LIN {X 0,Y 526.287,Z 607.372,A -85,B 0,C 180,E1 -4788.6,E2 -4788.6} C_VEL
LIN {X 0,Y 526.834,Z 594.37,A -85,B 0,C 180,E1 -4789.583,E2 -4789.583} C_VEL
LIN {X 0,Y 527.395,Z 580.497,A -85,B 0,C 180,E1 -4790.475,E2 -4790.475} C_VEL
LIN {X 0,Y 528.125,Z 564.209,A -85,B 0,C 180,E1 -4791.327,E2 -4791.327} C_VEL
LIN {X 0,Y 528.573,Z 550.297,A -85,B 0,C 180,E1 -4791.908,E2 -4791.908} C_VEL
LIN {X 0,Y 529.049,Z 533.497,A -85,B 0,C 180,E1 -4792.453,E2 -4792.453} C_VEL
LIN {X 0,Y 529.379,Z 517.227,A -85,B 0,C 180,E1 -4792.824,E2 -4792.824} C_VEL
LIN {X 0,Y 530.896,Z 327.244,A -85,B 0,C 180,E1 -4795.531,E2 -4795.531} C_VEL
LIN {X 0,Y 530.306,Z 322.417,A -85,B 0,C 180,E1 -4795.632,E2 -4795.632} C_VEL
LIN {X 0,Y 528.19,Z 310.861,A -85,B 0,C 180,E1 -4795.923,E2 -4795.923} C_VEL
LIN {X 0,Y 529.061,Z 286.972,A -85,B 0,C 180,E1 -4798.171,E2 -4798.171} C_VEL
LIN {X 0,Y 524.52,Z 271.582,A -85,B 0,C 180,E1 -4799.941,E2 -4799.941} C_VEL
LIN {X 0,Y 523.928,Z 269.536,A -85,B 0,C 180,E1 -4800.2,E2 -4800.2} C_VEL
LIN {X 0,Y 523.939,Z 269.532,A -85,B 0,C 180,E1 -4803.364,E2 -4803.364} C_VEL
LIN {X 0,Y 523.901,Z 269.535,A -85,B 0,C 180,E1 -4806.401,E2 -4806.401} C_VEL
LIN {X 0,Y 523.92,Z 269.539,A -85,B 0,C 180,E1 -4809.084,E2 -4809.084} C_VEL
LIN {X 0,Y 523.955,Z 269.527,A -85,B 0,C 180,E1 -4812.118,E2 -4812.118} C_VEL
LIN {X 0,Y 523.952,Z 269.534,A -85,B 0,C 180,E1 -4815.309,E2 -4815.309} C_VEL
LIN {X 0,Y 523.959,Z 269.526,A -85,B 0,C 180,E1 -4818.689,E2 -4818.689} C_VEL
LIN {X 0,Y 523.913,Z 269.531,A -85,B 0,C 180,E1 -4821.898,E2 -4821.898} C_VEL
LIN {X 0,Y 523.933,Z 269.533,A -85,B 0,C 180,E1 -4824.909,E2 -4824.909} C_VEL
LIN {X 0,Y 523.932,Z 269.532,A -85,B 0,C 180,E1 -4827.68,E2 -4827.68} C_VEL
LIN {X 0,Y 523.951,Z 269.528,A -85,B 0,C 180,E1 -4830.676,E2 -4830.676} C_VEL
LIN {X 0,Y 523.971,Z 269.527,A -85,B 0,C 180,E1 -4833.729,E2 -4833.729} C_VEL
LIN {X 0,Y 523.934,Z 269.529,A -85,B 0,C 180,E1 -4836.271,E2 -4836.271} C_VEL
LIN {X 0,Y 523.943,Z 269.531,A -85,B 0,C 180,E1 -4838.767,E2 -4838.767} C_VEL
LIN {X 0,Y 523.947,Z 269.53,A -85,B 0,C 180,E1 -4841.221,E2 -4841.221} C_VEL
LIN {X 0,Y 523.934,Z 269.531,A -85,B 0,C 180,E1 -4843.639,E2 -4843.639} C_VEL
LIN {X 0,Y 523.936,Z 269.521,A -85,B 0,C 180,E1 -4846.028,E2 -4846.028} C_VEL
LIN {X 0,Y 524.01,Z 269.518,A -85,B 0,C 180,E1 -4848.394,E2 -4848.394} C_VEL
LIN {X 0,Y 524.001,Z 269.52,A -85,B 0,C 180,E1 -4851.516,E2 -4851.516} C_VEL
LIN {X 0,Y 524.083,Z 269.505,A -85,B 0,C 180,E1 -4854.614,E2 -4854.614} C_VEL
LIN {X 0,Y 524.111,Z 269.508,A -85,B 0,C 180,E1 -4857.695,E2 -4857.695} C_VEL
LIN {X 0,Y 524.12,Z 269.503,A -85,B 0,C 180,E1 -4860.768,E2 -4860.768} C_VEL
LIN {X 0,Y 524.07,Z 269.518,A -85,B 0,C 180,E1 -4863.075,E2 -4863.075} C_VEL
LIN {X 0,Y 524.035,Z 269.515,A -85,B 0,C 180,E1 -4866.159,E2 -4866.159} C_VEL
LIN {X 0,Y 524.001,Z 269.512,A -85,B 0,C 180,E1 -4868.484,E2 -4868.484} C_VEL
LIN {X 0,Y 524.001,Z 269.522,A -85,B 0,C 180,E1 -4871.74,E2 -4871.74} C_VEL
LIN {X 0,Y 523.991,Z 269.52,A -85,B 0,C 180,E1 -4875.052,E2 -4875.052} C_VEL
LIN {X 0,Y 523.962,Z 269.526,A -85,B 0,C 180,E1 -4877.969,E2 -4877.969} C_VEL
LIN {X 0,Y 523.97,Z 269.525,A -85,B 0,C 180,E1 -4880.41,E2 -4880.41} C_VEL
LIN {X 0,Y 523.915,Z 269.532,A -85,B 0,C 180,E1 -4882.893,E2 -4882.893} C_VEL
LIN {X 0,Y 523.951,Z 269.529,A -85,B 0,C 180,E1 -4885.419,E2 -4885.419} C_VEL
LIN {X 0,Y 523.966,Z 269.517,A -85,B 0,C 180,E1 -4887.999,E2 -4887.999} C_VEL
LIN {X 0,Y 523.942,Z 269.537,A -85,B 0,C 180,E1 -4890.855,E2 -4890.855} C_VEL
LIN {X 0,Y 523.96,Z 269.526,A -85,B 0,C 180,E1 -4893.735,E2 -4893.735} C_VEL
LIN {X 0,Y 523.921,Z 269.533,A -85,B 0,C 180,E1 -4896.405,E2 -4896.405} C_VEL
LIN {X 0,Y 523.919,Z 269.536,A -85,B 0,C 180,E1 -4899.085,E2 -4899.085} C_VEL
LIN {X 0,Y 523.953,Z 269.524,A -85,B 0,C 180,E1 -4902.119,E2 -4902.119} C_VEL
LIN {X 0,Y 523.954,Z 269.525,A -85,B 0,C 180,E1 -4905.309,E2 -4905.309} C_VEL
LIN {X 0,Y 523.919,Z 269.536,A -85,B 0,C 180,E1 -4906.906,E2 -4906.906} C_VEL
LIN {X 0,Y 523.253,Z 269.617,A -85,B 0,C 180,E1 -4907.548,E2 -4907.548} C_VEL
LIN {X 0,Y 520.41,Z 269.975,A -85,B 0,C 180,E1 -4908.589,E2 -4908.589} C_VEL
LIN {X 0,Y 518.005,Z 270.272,A -85,B 0,C 180,E1 -4909.428,E2 -4909.428} C_VEL
LIN {X 0,Y 516.968,Z 270.4,A -85,B 0,C 180,E1 -4910.076,E2 -4910.076} C_VEL
LIN {X 0,Y 516.881,Z 270.411,A -85,B 0,C 180,E1 -4910.295,E2 -4910.295} C_VEL
LIN {X 0,Y 516.876,Z 270.406,A -85,B 0,C 180,E1 -4913.343,E2 -4913.343} C_VEL
LIN {X 0,Y 516.907,Z 270.406,A -85,B 0,C 180,E1 -4916.121,E2 -4916.121} C_VEL
LIN {X 0,Y 516.891,Z 270.413,A -85,B 0,C 180,E1 -4918.936,E2 -4918.936} C_VEL
LIN {X 0,Y 516.915,Z 270.446,A -85,B 0,C 180,E1 -4921.969,E2 -4921.969} C_VEL
LIN {X 0,Y 520.811,Z 284.241,A -85,B 0,C 180,E1 -4923.752,E2 -4923.752} C_VEL
LIN {X 0,Y 522.643,Z 289.186,A -85,B 0,C 180,E1 -4923.926,E2 -4923.926} C_VEL
LIN {X 0,Y 524.623,Z 299.71,A -85,B 0,C 180,E1 -4924.19,E2 -4924.19} C_VEL
LIN {X 0,Y 523.01,Z 486.351,A -85,B 0,C 180,E1 -4926.882,E2 -4926.882} C_VEL
LIN {X 0,Y 522.699,Z 501.745,A -85,B 0,C 180,E1 -4927.207,E2 -4927.207} C_VEL
LIN {X 0,Y 522.27,Z 516.651,A -85,B 0,C 180,E1 -4927.657,E2 -4927.657} C_VEL
LIN {X 0,Y 521.782,Z 530.861,A -85,B 0,C 180,E1 -4928.222,E2 -4928.222} C_VEL
LIN {X 0,Y 521.147,Z 545.811,A -85,B 0,C 180,E1 -4928.958,E2 -4928.958} C_VEL
LIN {X 0,Y 520.476,Z 560.69,A -85,B 0,C 180,E1 -4929.859,E2 -4929.859} C_VEL
LIN {X 0,Y 519.797,Z 574.326,A -85,B 0,C 180,E1 -4930.86,E2 -4930.86} C_VEL
LIN {X 0,Y 519.073,Z 588.127,A -85,B 0,C 180,E1 -4932.06,E2 -4932.06} C_VEL
LIN {X 0,Y 518.494,Z 599.871,A -85,B 0,C 180,E1 -4933.26,E2 -4933.26} C_VEL
LIN {X 0,Y 517.874,Z 611.317,A -85,B 0,C 180,E1 -4934.62,E2 -4934.62} C_VEL
LIN {X 0,Y 517.41,Z 621.483,A -85,B 0,C 180,E1 -4936.049,E2 -4936.049} C_VEL
LIN {X 0,Y 517.016,Z 631.096,A -85,B 0,C 180,E1 -4937.638,E2 -4937.638} C_VEL
LIN {X 0,Y 516.774,Z 638.267,A -85,B 0,C 180,E1 -4939.024,E2 -4939.024} C_VEL
LIN {X 0,Y 516.504,Z 645.083,A -85,B 0,C 180,E1 -4940.603,E2 -4940.603} C_VEL
LIN {X 0,Y 516.412,Z 650.683,A -85,B 0,C 180,E1 -4942.178,E2 -4942.178} C_VEL
LIN {X 0,Y 516.325,Z 655.19,A -85,B 0,C 180,E1 -4943.749,E2 -4943.749} C_VEL
LIN {X 0,Y 516.227,Z 658.571,A -85,B 0,C 180,E1 -4945.315,E2 -4945.315} C_VEL
LIN {X 0,Y 516.268,Z 661.031,A -85,B 0,C 180,E1 -4946.879,E2 -4946.879} C_VEL
LIN {X 0,Y 516.187,Z 662.449,A -85,B 0,C 180,E1 -4948.44,E2 -4948.44} C_VEL
LIN {X 0,Y 516.151,Z 662.997,A -85,B 0,C 180,E1 -4950,E2 -4950} C_VEL
LIN {X 0,Y 516.186,Z 662.505,A -85,B 0,C 180,E1 -4951.56,E2 -4951.56} C_VEL
LIN {X 0,Y 516.268,Z 661.142,A -85,B 0,C 180,E1 -4953.121,E2 -4953.121} C_VEL
LIN {X 0,Y 516.225,Z 658.736,A -85,B 0,C 180,E1 -4954.685,E2 -4954.685} C_VEL
LIN {X 0,Y 516.325,Z 655.423,A -85,B 0,C 180,E1 -4956.251,E2 -4956.251} C_VEL
LIN {X 0,Y 516.449,Z 649.731,A -85,B 0,C 180,E1 -4958.215,E2 -4958.215} C_VEL
LIN {X 0,Y 516.617,Z 642.247,A -85,B 0,C 180,E1 -4960.186,E2 -4960.186} C_VEL
LIN {X 0,Y 516.933,Z 634.612,A -85,B 0,C 180,E1 -4961.796,E2 -4961.796} C_VEL
LIN {X 0,Y 517.225,Z 625.828,A -85,B 0,C 180,E1 -4963.355,E2 -4963.355} C_VEL
LIN {X 0,Y 517.732,Z 615.185,A -85,B 0,C 180,E1 -4964.946,E2 -4964.946} C_VEL
LIN {X 0,Y 518.268,Z 604.197,A -85,B 0,C 180,E1 -4966.342,E2 -4966.342} C_VEL
LIN {X 0,Y 518.903,Z 591.185,A -85,B 0,C 180,E1 -4967.742,E2 -4967.742} C_VEL
LIN {X 0,Y 519.624,Z 577.891,A -85,B 0,C 180,E1 -4968.941,E2 -4968.941} C_VEL
LIN {X 0,Y 520.297,Z 564.794,A -85,B 0,C 180,E1 -4969.942,E2 -4969.942} C_VEL
LIN {X 0,Y 520.951,Z 550.864,A -85,B 0,C 180,E1 -4970.843,E2 -4970.843} C_VEL
LIN {X 0,Y 521.592,Z 535.502,A -85,B 0,C 180,E1 -4971.662,E2 -4971.662} C_VEL
LIN {X 0,Y 522.15,Z 520.391,A -85,B 0,C 180,E1 -4972.296,E2 -4972.296} C_VEL
LIN {X 0,Y 522.607,Z 503.979,A -85,B 0,C 180,E1 -4972.823,E2 -4972.823} C_VEL
LIN {X 0,Y 522.95,Z 487.016,A -85,B 0,C 180,E1 -4973.199,E2 -4973.199} C_VEL
LIN {X 0,Y 524.614,Z 299.802,A -85,B 0,C 180,E1 -4975.899,E2 -4975.899} C_VEL
LIN {X 0,Y 522.346,Z 287.999,A -85,B 0,C 180,E1 -4976.198,E2 -4976.198} C_VEL
LIN {X 0,Y 520.74,Z 284.073,A -85,B 0,C 180,E1 -4976.357,E2 -4976.357} C_VEL
LIN {X 0,Y 516.91,Z 270.411,A -85,B 0,C 180,E1 -4978.158,E2 -4978.158} C_VEL
LIN {X 0,Y 516.888,Z 270.416,A -85,B 0,C 180,E1 -4981.109,E2 -4981.109} C_VEL
LIN {X 0,Y 516.906,Z 270.41,A -85,B 0,C 180,E1 -4983.966,E2 -4983.966} C_VEL
LIN {X 0,Y 516.852,Z 270.406,A -85,B 0,C 180,E1 -4986.748,E2 -4986.748} C_VEL
LIN {X 0,Y 516.88,Z 270.411,A -85,B 0,C 180,E1 -4989.721,E2 -4989.721} C_VEL
LIN {X 0,Y 516.911,Z 270.405,A -85,B 0,C 180,E1 -4991.775,E2 -4991.775} C_VEL
LIN {X 0,Y 516.921,Z 270.409,A -85,B 0,C 180,E1 -4995.01,E2 -4995.01} C_VEL
LIN {X 0,Y 516.913,Z 270.403,A -85,B 0,C 180,E1 -4998.398,E2 -4998.398} C_VEL
LIN {X 0,Y 516.879,Z 270.415,A -85,B 0,C 180,E1 -5001.284,E2 -5001.284} C_VEL
LIN {X 0,Y 516.886,Z 270.407,A -85,B 0,C 180,E1 -5004.221,E2 -5004.221} C_VEL
LIN {X 0,Y 516.893,Z 270.409,A -85,B 0,C 180,E1 -5007.053,E2 -5007.053} C_VEL
LIN {X 0,Y 516.89,Z 270.408,A -85,B 0,C 180,E1 -5009.796,E2 -5009.796} C_VEL
LIN {X 0,Y 516.923,Z 270.397,A -85,B 0,C 180,E1 -5012.467,E2 -5012.467} C_VEL
LIN {X 0,Y 516.908,Z 270.412,A -85,B 0,C 180,E1 -5015.072,E2 -5015.072} C_VEL
LIN {X 0,Y 516.867,Z 270.404,A -85,B 0,C 180,E1 -5017.621,E2 -5017.621} C_VEL
LIN {X 0,Y 516.929,Z 270.402,A -85,B 0,C 180,E1 -5020.13,E2 -5020.13} C_VEL
LIN {X 0,Y 516.918,Z 270.404,A -85,B 0,C 180,E1 -5022.596,E2 -5022.596} C_VEL
LIN {X 0,Y 516.939,Z 270.4,A -85,B 0,C 180,E1 -5025.03,E2 -5025.03} C_VEL
LIN {X 0,Y 516.963,Z 270.397,A -85,B 0,C 180,E1 -5028.234,E2 -5028.234} C_VEL
LIN {X 0,Y 516.963,Z 270.399,A -85,B 0,C 180,E1 -5031.399,E2 -5031.399} C_VEL
LIN {X 0,Y 517.013,Z 270.392,A -85,B 0,C 180,E1 -5033.757,E2 -5033.757} C_VEL
LIN {X 0,Y 517.082,Z 270.378,A -85,B 0,C 180,E1 -5037.663,E2 -5037.663} C_VEL
LIN {X 0,Y 517.091,Z 270.388,A -85,B 0,C 180,E1 -5040.779,E2 -5040.779} C_VEL
LIN {X 0,Y 517.01,Z 270.388,A -85,B 0,C 180,E1 -5043.117,E2 -5043.117} C_VEL
LIN {X 0,Y 517.013,Z 270.391,A -85,B 0,C 180,E1 -5046.243,E2 -5046.243} C_VEL
LIN {X 0,Y 516.949,Z 270.396,A -85,B 0,C 180,E1 -5049.389,E2 -5049.389} C_VEL
LIN {X 0,Y 516.949,Z 270.396,A -85,B 0,C 180,E1 -5051.807,E2 -5051.807} C_VEL
LIN {X 0,Y 516.941,Z 270.406,A -85,B 0,C 180,E1 -5055.146,E2 -5055.146} C_VEL
LIN {X 0,Y 516.922,Z 270.403,A -85,B 0,C 180,E1 -5058.222,E2 -5058.222} C_VEL
LIN {X 0,Y 516.909,Z 270.412,A -85,B 0,C 180,E1 -5060.701,E2 -5060.701} C_VEL
LIN {X 0,Y 516.908,Z 270.405,A -85,B 0,C 180,E1 -5064.072,E2 -5064.072} C_VEL
LIN {X 0,Y 516.921,Z 270.411,A -85,B 0,C 180,E1 -5066.658,E2 -5066.658} C_VEL
LIN {X 0,Y 516.908,Z 270.406,A -85,B 0,C 180,E1 -5069.524,E2 -5069.524} C_VEL
LIN {X 0,Y 516.894,Z 270.414,A -85,B 0,C 180,E1 -5072.544,E2 -5072.544} C_VEL
LIN {X 0,Y 516.88,Z 270.411,A -85,B 0,C 180,E1 -5075.332,E2 -5075.332} C_VEL
LIN {X 0,Y 516.878,Z 270.411,A -85,B 0,C 180,E1 -5077.943,E2 -5077.943} C_VEL
LIN {X 0,Y 516.883,Z 270.418,A -85,B 0,C 180,E1 -5080.741,E2 -5080.741} C_VEL
LIN {X 0,Y 516.88,Z 270.418,A -85,B 0,C 180,E1 -5082.831,E2 -5082.831} C_VEL
LIN {X 0,Y 516.92,Z 270.41,A -85,B 0,C 180,E1 -5085.01,E2 -5085.01} C_VEL
LIN {X 0,Y 516.915,Z 270.41,A -85,B 0,C 180,E1 -5088.398,E2 -5088.398} C_VEL
LIN {X 0,Y 516.879,Z 270.412,A -85,B 0,C 180,E1 -5091.284,E2 -5091.284} C_VEL
LIN {X 0,Y 516.868,Z 270.415,A -85,B 0,C 180,E1 -5094.22,E2 -5094.22} C_VEL
LIN {X 0,Y 516.892,Z 270.412,A -85,B 0,C 180,E1 -5097.053,E2 -5097.053} C_VEL
LIN {X 0,Y 516.929,Z 270.524,A -85,B 0,C 180,E1 -5099.489,E2 -5099.489} C_VEL
LIN {X 0,Y 522.347,Z 288.675,A -85,B 0,C 180,E1 -5101.621,E2 -5101.621} C_VEL
LIN {X 0,Y 521.529,Z 310.726,A -85,B 0,C 180,E1 -5103.729,E2 -5103.729} C_VEL
LIN {X 0,Y 524.483,Z 326.998,A -85,B 0,C 180,E1 -5104.134,E2 -5104.134} C_VEL
LIN {X 0,Y 522.827,Z 517.021,A -85,B 0,C 180,E1 -5106.873,E2 -5106.873} C_VEL
LIN {X 0,Y 522.51,Z 532.367,A -85,B 0,C 180,E1 -5107.225,E2 -5107.225} C_VEL
LIN {X 0,Y 521.971,Z 548.783,A -85,B 0,C 180,E1 -5107.748,E2 -5107.748} C_VEL
LIN {X 0,Y 521.453,Z 563.992,A -85,B 0,C 180,E1 -5108.385,E2 -5108.385} C_VEL
LIN {X 0,Y 520.681,Z 580.296,A -85,B 0,C 180,E1 -5109.249,E2 -5109.249} C_VEL
LIN {X 0,Y 520.003,Z 595.596,A -85,B 0,C 180,E1 -5110.252,E2 -5110.252} C_VEL
LIN {X 0,Y 519.341,Z 609.107,A -85,B 0,C 180,E1 -5111.311,E2 -5111.311} C_VEL
LIN {X 0,Y 518.724,Z 621.594,A -85,B 0,C 180,E1 -5112.455,E2 -5112.455} C_VEL
LIN {X 0,Y 518.148,Z 632.841,A -85,B 0,C 180,E1 -5113.654,E2 -5113.654} C_VEL
LIN {X 0,Y 517.703,Z 642.621,A -85,B 0,C 180,E1 -5114.859,E2 -5114.859} C_VEL
LIN {X 0,Y 517.296,Z 652.452,A -85,B 0,C 180,E1 -5116.246,E2 -5116.246} C_VEL
LIN {X 0,Y 516.945,Z 661.963,A -85,B 0,C 180,E1 -5117.836,E2 -5117.836} C_VEL
LIN {X 0,Y 516.679,Z 669.919,A -85,B 0,C 180,E1 -5119.419,E2 -5119.419} C_VEL
LIN {X 0,Y 516.469,Z 676.56,A -85,B 0,C 180,E1 -5120.997,E2 -5120.997} C_VEL
LIN {X 0,Y 516.388,Z 681.949,A -85,B 0,C 180,E1 -5122.571,E2 -5122.571} C_VEL
LIN {X 0,Y 516.322,Z 685.25,A -85,B 0,C 180,E1 -5123.749,E2 -5123.749} C_VEL
LIN {X 0,Y 516.225,Z 688.633,A -85,B 0,C 180,E1 -5125.315,E2 -5125.315} C_VEL
LIN {X 0,Y 516.267,Z 691.091,A -85,B 0,C 180,E1 -5126.879,E2 -5126.879} C_VEL
LIN {X 0,Y 516.186,Z 692.477,A -85,B 0,C 180,E1 -5128.44,E2 -5128.44} C_VEL
LIN {X 0,Y 516.149,Z 693,A -85,B 0,C 180,E1 -5130,E2 -5130} C_VEL
LIN {X 0,Y 516.186,Z 692.477,A -85,B 0,C 180,E1 -5131.56,E2 -5131.56} C_VEL
LIN {X 0,Y 516.267,Z 691.089,A -85,B 0,C 180,E1 -5133.121,E2 -5133.121} C_VEL
LIN {X 0,Y 516.225,Z 688.632,A -85,B 0,C 180,E1 -5134.685,E2 -5134.685} C_VEL
LIN {X 0,Y 516.368,Z 684.558,A -85,B 0,C 180,E1 -5136.507,E2 -5136.507} C_VEL
LIN {X 0,Y 516.418,Z 679.433,A -85,B 0,C 180,E1 -5138.215,E2 -5138.215} C_VEL
LIN {X 0,Y 516.591,Z 671.742,A -85,B 0,C 180,E1 -5140.187,E2 -5140.187} C_VEL
LIN {X 0,Y 516.933,Z 663.169,A -85,B 0,C 180,E1 -5141.946,E2 -5141.946} C_VEL
LIN {X 0,Y 517.223,Z 653.697,A -85,B 0,C 180,E1 -5143.556,E2 -5143.556} C_VEL
LIN {X 0,Y 517.666,Z 644.064,A -85,B 0,C 180,E1 -5144.948,E2 -5144.948} C_VEL
LIN {X 0,Y 518.148,Z 632.839,A -85,B 0,C 180,E1 -5146.346,E2 -5146.346} C_VEL
LIN {X 0,Y 518.798,Z 620.611,A -85,B 0,C 180,E1 -5147.644,E2 -5147.644} C_VEL
LIN {X 0,Y 519.441,Z 607.562,A -85,B 0,C 180,E1 -5148.819,E2 -5148.819} C_VEL
LIN {X 0,Y 520.075,Z 594.16,A -85,B 0,C 180,E1 -5149.848,E2 -5149.848} C_VEL
LIN {X 0,Y 520.68,Z 580.288,A -85,B 0,C 180,E1 -5150.751,E2 -5150.751} C_VEL
LIN {X 0,Y 521.403,Z 565.136,A -85,B 0,C 180,E1 -5151.558,E2 -5151.558} C_VEL
LIN {X 0,Y 521.954,Z 550.088,A -85,B 0,C 180,E1 -5152.201,E2 -5152.201} C_VEL
LIN {X 0,Y 522.461,Z 533.288,A -85,B 0,C 180,E1 -5152.751,E2 -5152.751} C_VEL
LIN {X 0,Y 522.836,Z 517.019,A -85,B 0,C 180,E1 -5153.126,E2 -5153.126} C_VEL
LIN {X 0,Y 524.471,Z 328.39,A -85,B 0,C 180,E1 -5155.846,E2 -5155.846} C_VEL
LIN {X 0,Y 523.75,Z 322.787,A -85,B 0,C 180,E1 -5155.967,E2 -5155.967} C_VEL
LIN {X 0,Y 521.56,Z 310.77,A -85,B 0,C 180,E1 -5156.265,E2 -5156.265} C_VEL
LIN {X 0,Y 522.302,Z 288.658,A -85,B 0,C 180,E1 -5158.383,E2 -5158.383} C_VEL
LIN {X 0,Y 516.913,Z 270.411,A -85,B 0,C 180,E1 -5160.541,E2 -5160.541} C_VEL
LIN {X 0,Y 516.905,Z 270.41,A -85,B 0,C 180,E1 -5163.879,E2 -5163.879} C_VEL
LIN {X 0,Y 516.874,Z 270.412,A -85,B 0,C 180,E1 -5166.746,E2 -5166.746} C_VEL
LIN {X 0,Y 516.88,Z 270.413,A -85,B 0,C 180,E1 -5169.721,E2 -5169.721} C_VEL
LIN {X 0,Y 516.904,Z 270.408,A -85,B 0,C 180,E1 -5172.761,E2 -5172.761} C_VEL
LIN {X 0,Y 516.92,Z 270.407,A -85,B 0,C 180,E1 -5175.01,E2 -5175.01} C_VEL
LIN {X 0,Y 516.915,Z 270.402,A -85,B 0,C 180,E1 -5178.398,E2 -5178.398} C_VEL
LIN {X 0,Y 516.878,Z 270.415,A -85,B 0,C 180,E1 -5181.284,E2 -5181.284} C_VEL
LIN {X 0,Y 516.885,Z 270.406,A -85,B 0,C 180,E1 -5184.221,E2 -5184.221} C_VEL
LIN {X 0,Y 516.892,Z 270.413,A -85,B 0,C 180,E1 -5187.053,E2 -5187.053} C_VEL
LIN {X 0,Y 516.889,Z 270.407,A -85,B 0,C 180,E1 -5189.796,E2 -5189.796} C_VEL
LIN {X 0,Y 516.923,Z 270.403,A -85,B 0,C 180,E1 -5192.467,E2 -5192.467} C_VEL
LIN {X 0,Y 516.908,Z 270.412,A -85,B 0,C 180,E1 -5195.072,E2 -5195.072} C_VEL
LIN {X 0,Y 516.867,Z 270.411,A -85,B 0,C 180,E1 -5197.622,E2 -5197.622} C_VEL
LIN {X 0,Y 516.928,Z 270.393,A -85,B 0,C 180,E1 -5200.13,E2 -5200.13} C_VEL
LIN {X 0,Y 516.918,Z 270.404,A -85,B 0,C 180,E1 -5202.596,E2 -5202.596} C_VEL
LIN {X 0,Y 516.939,Z 270.403,A -85,B 0,C 180,E1 -5205.03,E2 -5205.03} C_VEL
LIN {X 0,Y 516.963,Z 270.395,A -85,B 0,C 180,E1 -5208.234,E2 -5208.234} C_VEL
LIN {X 0,Y 516.966,Z 270.398,A -85,B 0,C 180,E1 -5211.4,E2 -5211.4} C_VEL
LIN {X 0,Y 517.013,Z 270.384,A -85,B 0,C 180,E1 -5213.757,E2 -5213.757} C_VEL
LIN {X 0,Y 517.083,Z 270.384,A -85,B 0,C 180,E1 -5217.663,E2 -5217.663} C_VEL
LIN {X 0,Y 517.091,Z 270.377,A -85,B 0,C 180,E1 -5220.779,E2 -5220.779} C_VEL
LIN {X 0,Y 517.011,Z 270.397,A -85,B 0,C 180,E1 -5223.117,E2 -5223.117} C_VEL
LIN {X 0,Y 517,Z 270.392,A -85,B 0,C 180,E1 -5226.243,E2 -5226.243} C_VEL
LIN {X 0,Y 516.95,Z 270.4,A -85,B 0,C 180,E1 -5229.389,E2 -5229.389} C_VEL
LIN {X 0,Y 516.95,Z 270.4,A -85,B 0,C 180,E1 -5231.807,E2 -5231.807} C_VEL
LIN {X 0,Y 516.942,Z 270.397,A -85,B 0,C 180,E1 -5235.147,E2 -5235.147} C_VEL
LIN {X 0,Y 516.923,Z 270.403,A -85,B 0,C 180,E1 -5238.222,E2 -5238.222} C_VEL
LIN {X 0,Y 516.91,Z 270.408,A -85,B 0,C 180,E1 -5240.702,E2 -5240.702} C_VEL
LIN {X 0,Y 516.91,Z 270.404,A -85,B 0,C 180,E1 -5244.072,E2 -5244.072} C_VEL
LIN {X 0,Y 516.922,Z 270.407,A -85,B 0,C 180,E1 -5246.658,E2 -5246.658} C_VEL
LIN {X 0,Y 516.909,Z 270.405,A -85,B 0,C 180,E1 -5249.524,E2 -5249.524} C_VEL
LIN {X 0,Y 516.894,Z 270.409,A -85,B 0,C 180,E1 -5252.544,E2 -5252.544} C_VEL
LIN {X 0,Y 516.882,Z 270.41,A -85,B 0,C 180,E1 -5255.333,E2 -5255.333} C_VEL
LIN {X 0,Y 516.879,Z 270.402,A -85,B 0,C 180,E1 -5257.943,E2 -5257.943} C_VEL
LIN {X 0,Y 516.882,Z 270.415,A -85,B 0,C 180,E1 -5260.742,E2 -5260.742} C_VEL
LIN {X 0,Y 516.883,Z 270.41,A -85,B 0,C 180,E1 -5262.832,E2 -5262.832} C_VEL
LIN {X 0,Y 516.922,Z 270.405,A -85,B 0,C 180,E1 -5265.01,E2 -5265.01} C_VEL
LIN {X 0,Y 516.917,Z 270.408,A -85,B 0,C 180,E1 -5268.398,E2 -5268.398} C_VEL
LIN {X 0,Y 516.881,Z 270.411,A -85,B 0,C 180,E1 -5270.295,E2 -5270.295} C_VEL
LIN {X 0,Y 516.211,Z 270.498,A -85,B 0,C 180,E1 -5270.945,E2 -5270.945} C_VEL
LIN {X 0,Y 513.364,Z 270.849,A -85,B 0,C 180,E1 -5272.001,E2 -5272.001} C_VEL
LIN {X 0,Y 510.954,Z 271.147,A -85,B 0,C 180,E1 -5272.851,E2 -5272.851} C_VEL
LIN {X 0,Y 509.91,Z 271.275,A -85,B 0,C 180,E1 -5273.508,E2 -5273.508} C_VEL
LIN {X 0,Y 509.819,Z 271.286,A -85,B 0,C 180,E1 -5273.73,E2 -5273.73} C_VEL
LIN {X 0,Y 509.858,Z 271.281,A -85,B 0,C 180,E1 -5276.539,E2 -5276.539} C_VEL
LIN {X 0,Y 509.845,Z 271.289,A -85,B 0,C 180,E1 -5279.334,E2 -5279.334} C_VEL
LIN {X 0,Y 509.874,Z 271.292,A -85,B 0,C 180,E1 -5281.622,E2 -5281.622} C_VEL
LIN {X 0,Y 513.597,Z 284.347,A -85,B 0,C 180,E1 -5283.345,E2 -5283.345} C_VEL
LIN {X 0,Y 516.417,Z 291.107,A -85,B 0,C 180,E1 -5283.613,E2 -5283.613} C_VEL
LIN {X 0,Y 518.215,Z 299.803,A -85,B 0,C 180,E1 -5283.845,E2 -5283.845} C_VEL
LIN {X 0,Y 516.486,Z 486.597,A -85,B 0,C 180,E1 -5286.573,E2 -5286.573} C_VEL
LIN {X 0,Y 516.175,Z 501.975,A -85,B 0,C 180,E1 -5286.903,E2 -5286.903} C_VEL
LIN {X 0,Y 515.669,Z 518.364,A -85,B 0,C 180,E1 -5287.408,E2 -5287.408} C_VEL
LIN {X 0,Y 515.086,Z 533.568,A -85,B 0,C 180,E1 -5288.041,E2 -5288.041} C_VEL
LIN {X 0,Y 514.422,Z 547.787,A -85,B 0,C 180,E1 -5288.775,E2 -5288.775} C_VEL
LIN {X 0,Y 513.801,Z 560.908,A -85,B 0,C 180,E1 -5289.586,E2 -5289.586} C_VEL
LIN {X 0,Y 513.05,Z 574.543,A -85,B 0,C 180,E1 -5290.599,E2 -5290.599} C_VEL
LIN {X 0,Y 512.31,Z 587.281,A -85,B 0,C 180,E1 -5291.711,E2 -5291.711} C_VEL
LIN {X 0,Y 511.618,Z 600.086,A -85,B 0,C 180,E1 -5293.028,E2 -5293.028} C_VEL
LIN {X 0,Y 510.943,Z 612.03,A -85,B 0,C 180,E1 -5294.474,E2 -5294.474} C_VEL
LIN {X 0,Y 510.401,Z 623.036,A -85,B 0,C 180,E1 -5296.056,E2 -5296.056} C_VEL
LIN {X 0,Y 509.978,Z 632.414,A -85,B 0,C 180,E1 -5297.666,E2 -5297.666} C_VEL
LIN {X 0,Y 509.689,Z 640.268,A -85,B 0,C 180,E1 -5299.272,E2 -5299.272} C_VEL
LIN {X 0,Y 509.44,Z 646.824,A -85,B 0,C 180,E1 -5300.872,E2 -5300.872} C_VEL
LIN {X 0,Y 509.329,Z 652.122,A -85,B 0,C 180,E1 -5302.468,E2 -5302.468} C_VEL
LIN {X 0,Y 509.258,Z 655.4,A -85,B 0,C 180,E1 -5303.661,E2 -5303.661} C_VEL
LIN {X 0,Y 509.145,Z 658.779,A -85,B 0,C 180,E1 -5305.249,E2 -5305.249} C_VEL
LIN {X 0,Y 509.185,Z 661.232,A -85,B 0,C 180,E1 -5306.835,E2 -5306.835} C_VEL
LIN {X 0,Y 509.108,Z 662.634,A -85,B 0,C 180,E1 -5308.418,E2 -5308.418} C_VEL
LIN {X 0,Y 509.062,Z 663.177,A -85,B 0,C 180,E1 -5310,E2 -5310} C_VEL
LIN {X 0,Y 509.107,Z 662.689,A -85,B 0,C 180,E1 -5311.582,E2 -5311.582} C_VEL
LIN {X 0,Y 509.185,Z 661.34,A -85,B 0,C 180,E1 -5313.165,E2 -5313.165} C_VEL
LIN {X 0,Y 509.143,Z 658.943,A -85,B 0,C 180,E1 -5314.751,E2 -5314.751} C_VEL
LIN {X 0,Y 509.307,Z 655.16,A -85,B 0,C 180,E1 -5316.517,E2 -5316.517} C_VEL
LIN {X 0,Y 509.373,Z 649.938,A -85,B 0,C 180,E1 -5318.33,E2 -5318.33} C_VEL
LIN {X 0,Y 509.593,Z 642.453,A -85,B 0,C 180,E1 -5320.328,E2 -5320.328} C_VEL
LIN {X 0,Y 509.938,Z 633.967,A -85,B 0,C 180,E1 -5322.133,E2 -5322.133} C_VEL
LIN {X 0,Y 510.326,Z 624.812,A -85,B 0,C 180,E1 -5323.742,E2 -5323.742} C_VEL
LIN {X 0,Y 510.859,Z 614.114,A -85,B 0,C 180,E1 -5325.329,E2 -5325.329} C_VEL
LIN {X 0,Y 511.465,Z 602.632,A -85,B 0,C 180,E1 -5326.772,E2 -5326.772} C_VEL
LIN {X 0,Y 512.139,Z 590.331,A -85,B 0,C 180,E1 -5328.088,E2 -5328.088} C_VEL
LIN {X 0,Y 512.955,Z 576.92,A -85,B 0,C 180,E1 -5329.301,E2 -5329.301} C_VEL
LIN {X 0,Y 513.665,Z 563.574,A -85,B 0,C 180,E1 -5330.315,E2 -5330.315} C_VEL
LIN {X 0,Y 514.384,Z 549.303,A -85,B 0,C 180,E1 -5331.227,E2 -5331.227} C_VEL
LIN {X 0,Y 515.01,Z 534.571,A -85,B 0,C 180,E1 -5332.006,E2 -5332.006} C_VEL
LIN {X 0,Y 515.657,Z 519.284,A -85,B 0,C 180,E1 -5332.645,E2 -5332.645} C_VEL
LIN {X 0,Y 516.114,Z 503.248,A -85,B 0,C 180,E1 -5333.153,E2 -5333.153} C_VEL
LIN {X 0,Y 516.452,Z 487.185,A -85,B 0,C 180,E1 -5333.509,E2 -5333.509} C_VEL
LIN {X 0,Y 518.236,Z 301.157,A -85,B 0,C 180,E1 -5336.224,E2 -5336.224} C_VEL
LIN {X 0,Y 516.688,Z 292.333,A -85,B 0,C 180,E1 -5336.443,E2 -5336.443} C_VEL
LIN {X 0,Y 515.51,Z 288.822,A -85,B 0,C 180,E1 -5336.562,E2 -5336.562} C_VEL
LIN {X 0,Y 513.56,Z 284.267,A -85,B 0,C 180,E1 -5336.756,E2 -5336.756} C_VEL
LIN {X 0,Y 509.881,Z 271.287,A -85,B 0,C 180,E1 -5338.487,E2 -5338.487} C_VEL
LIN {X 0,Y 509.819,Z 271.295,A -85,B 0,C 180,E1 -5341.59,E2 -5341.59} C_VEL
LIN {X 0,Y 509.846,Z 271.289,A -85,B 0,C 180,E1 -5344.414,E2 -5344.414} C_VEL
LIN {X 0,Y 509.807,Z 271.289,A -85,B 0,C 180,E1 -5347.341,E2 -5347.341} C_VEL
LIN {X 0,Y 509.837,Z 271.285,A -85,B 0,C 180,E1 -5350.382,E2 -5350.382} C_VEL
LIN {X 0,Y 509.824,Z 271.29,A -85,B 0,C 180,E1 -5353.062,E2 -5353.062} C_VEL
LIN {X 0,Y 509.829,Z 271.287,A -85,B 0,C 180,E1 -5355.792,E2 -5355.792} C_VEL
LIN {X 0,Y 509.855,Z 271.284,A -85,B 0,C 180,E1 -5358.574,E2 -5358.574} C_VEL
LIN {X 0,Y 509.849,Z 271.284,A -85,B 0,C 180,E1 -5361.786,E2 -5361.786} C_VEL
LIN {X 0,Y 509.841,Z 271.286,A -85,B 0,C 180,E1 -5364.623,E2 -5364.623} C_VEL
LIN {X 0,Y 509.859,Z 271.284,A -85,B 0,C 180,E1 -5367.481,E2 -5367.481} C_VEL
LIN {X 0,Y 509.856,Z 271.284,A -85,B 0,C 180,E1 -5370.273,E2 -5370.273} C_VEL
LIN {X 0,Y 509.881,Z 271.278,A -85,B 0,C 180,E1 -5372.944,E2 -5372.944} C_VEL
LIN {X 0,Y 509.868,Z 271.284,A -85,B 0,C 180,E1 -5375.574,E2 -5375.574} C_VEL
LIN {X 0,Y 509.847,Z 271.283,A -85,B 0,C 180,E1 -5378.998,E2 -5378.998} C_VEL
LIN {X 0,Y 509.879,Z 271.279,A -85,B 0,C 180,E1 -5382.001,E2 -5382.001} C_VEL
LIN {X 0,Y 509.908,Z 271.272,A -85,B 0,C 180,E1 -5384.819,E2 -5384.819} C_VEL
LIN {X 0,Y 509.898,Z 271.277,A -85,B 0,C 180,E1 -5388.124,E2 -5388.124} C_VEL
LIN {X 0,Y 509.909,Z 271.277,A -85,B 0,C 180,E1 -5391.28,E2 -5391.28} C_VEL
LIN {X 0,Y 509.98,Z 271.269,A -85,B 0,C 180,E1 -5393.67,E2 -5393.67} C_VEL
LIN {X 0,Y 510.053,Z 271.253,A -85,B 0,C 180,E1 -5397.631,E2 -5397.631} C_VEL
LIN {X 0,Y 510.061,Z 271.263,A -85,B 0,C 180,E1 -5400.789,E2 -5400.789} C_VEL
LIN {X 0,Y 509.952,Z 271.266,A -85,B 0,C 180,E1 -5403.16,E2 -5403.16} C_VEL
LIN {X 0,Y 509.98,Z 271.267,A -85,B 0,C 180,E1 -5406.329,E2 -5406.329} C_VEL
LIN {X 0,Y 509.912,Z 271.282,A -85,B 0,C 180,E1 -5408.72,E2 -5408.72} C_VEL
LIN {X 0,Y 509.901,Z 271.274,A -85,B 0,C 180,E1 -5411.932,E2 -5411.932} C_VEL
LIN {X 0,Y 509.891,Z 271.283,A -85,B 0,C 180,E1 -5415.242,E2 -5415.242} C_VEL
LIN {X 0,Y 509.885,Z 271.279,A -85,B 0,C 180,E1 -5418.001,E2 -5418.001} C_VEL
LIN {X 0,Y 509.847,Z 271.29,A -85,B 0,C 180,E1 -5421.002,E2 -5421.002} C_VEL
LIN {X 0,Y 509.867,Z 271.285,A -85,B 0,C 180,E1 -5424.426,E2 -5424.426} C_VEL
LIN {X 0,Y 509.88,Z 271.286,A -85,B 0,C 180,E1 -5427.056,E2 -5427.056} C_VEL
LIN {X 0,Y 509.854,Z 271.284,A -85,B 0,C 180,E1 -5429.751,E2 -5429.751} C_VEL
LIN {X 0,Y 509.871,Z 271.289,A -85,B 0,C 180,E1 -5432.774,E2 -5432.774} C_VEL
LIN {X 0,Y 509.84,Z 271.286,A -85,B 0,C 180,E1 -5435.581,E2 -5435.581} C_VEL
LIN {X 0,Y 509.847,Z 271.29,A -85,B 0,C 180,E1 -5438.338,E2 -5438.338} C_VEL
LIN {X 0,Y 509.856,Z 271.287,A -85,B 0,C 180,E1 -5441.425,E2 -5441.425} C_VEL
LIN {X 0,Y 509.854,Z 271.293,A -85,B 0,C 180,E1 -5444.668,E2 -5444.668} C_VEL
LIN {X 0,Y 509.858,Z 271.286,A -85,B 0,C 180,E1 -5448.103,E2 -5448.103} C_VEL
LIN {X 0,Y 509.844,Z 271.293,A -85,B 0,C 180,E1 -5450.648,E2 -5450.648} C_VEL
LIN {X 0,Y 509.822,Z 271.29,A -85,B 0,C 180,E1 -5453.647,E2 -5453.647} C_VEL
LIN {X 0,Y 509.856,Z 271.285,A -85,B 0,C 180,E1 -5456.539,E2 -5456.539} C_VEL
LIN {X 0,Y 509.894,Z 271.437,A -85,B 0,C 180,E1 -5459.137,E2 -5459.137} C_VEL
LIN {X 0,Y 515.521,Z 290.215,A -85,B 0,C 180,E1 -5461.385,E2 -5461.385} C_VEL
LIN {X 0,Y 515.664,Z 293.613,A -85,B 0,C 180,E1 -5461.731,E2 -5461.731} C_VEL
LIN {X 0,Y 514.931,Z 310.628,A -85,B 0,C 180,E1 -5463.373,E2 -5463.373} C_VEL
LIN {X 0,Y 518.083,Z 328.672,A -85,B 0,C 180,E1 -5463.819,E2 -5463.819} C_VEL
LIN {X 0,Y 516.301,Z 516.813,A -85,B 0,C 180,E1 -5466.564,E2 -5466.564} C_VEL
LIN {X 0,Y 515.936,Z 532.159,A -85,B 0,C 180,E1 -5466.918,E2 -5466.918} C_VEL
LIN {X 0,Y 515.388,Z 548.575,A -85,B 0,C 180,E1 -5467.448,E2 -5467.448} C_VEL
LIN {X 0,Y 514.798,Z 564.105,A -85,B 0,C 180,E1 -5468.108,E2 -5468.108} C_VEL
LIN {X 0,Y 514.002,Z 580.087,A -85,B 0,C 180,E1 -5468.966,E2 -5468.966} C_VEL
LIN {X 0,Y 513.241,Z 595.386,A -85,B 0,C 180,E1 -5469.981,E2 -5469.981} C_VEL
LIN {X 0,Y 512.579,Z 607.838,A -85,B 0,C 180,E1 -5470.962,E2 -5470.962} C_VEL
LIN {X 0,Y 511.92,Z 620.402,A -85,B 0,C 180,E1 -5472.111,E2 -5472.111} C_VEL
LIN {X 0,Y 511.214,Z 632.63,A -85,B 0,C 180,E1 -5473.426,E2 -5473.426} C_VEL
LIN {X 0,Y 510.687,Z 643.852,A -85,B 0,C 180,E1 -5474.843,E2 -5474.843} C_VEL
LIN {X 0,Y 510.152,Z 654.727,A -85,B 0,C 180,E1 -5476.456,E2 -5476.456} C_VEL
LIN {X 0,Y 509.826,Z 664.36,A -85,B 0,C 180,E1 -5478.163,E2 -5478.163} C_VEL
LIN {X 0,Y 509.538,Z 671.533,A -85,B 0,C 180,E1 -5479.671,E2 -5479.671} C_VEL
LIN {X 0,Y 509.352,Z 679.222,A -85,B 0,C 180,E1 -5481.67,E2 -5481.67} C_VEL
LIN {X 0,Y 509.255,Z 685.071,A -85,B 0,C 180,E1 -5483.661,E2 -5483.661} C_VEL
LIN {X 0,Y 509.142,Z 688.49,A -85,B 0,C 180,E1 -5485.249,E2 -5485.249} C_VEL
LIN {X 0,Y 509.184,Z 690.978,A -85,B 0,C 180,E1 -5486.835,E2 -5486.835} C_VEL
LIN {X 0,Y 509.106,Z 692.379,A -85,B 0,C 180,E1 -5488.418,E2 -5488.418} C_VEL
LIN {X 0,Y 509.061,Z 692.906,A -85,B 0,C 180,E1 -5490,E2 -5490} C_VEL
LIN {X 0,Y 509.106,Z 692.378,A -85,B 0,C 180,E1 -5491.582,E2 -5491.582} C_VEL
LIN {X 0,Y 509.184,Z 690.977,A -85,B 0,C 180,E1 -5493.165,E2 -5493.165} C_VEL
LIN {X 0,Y 509.142,Z 688.49,A -85,B 0,C 180,E1 -5494.751,E2 -5494.751} C_VEL
LIN {X 0,Y 509.264,Z 684.7,A -85,B 0,C 180,E1 -5496.477,E2 -5496.477} C_VEL
LIN {X 0,Y 509.353,Z 679.225,A -85,B 0,C 180,E1 -5498.33,E2 -5498.33} C_VEL
LIN {X 0,Y 509.538,Z 671.533,A -85,B 0,C 180,E1 -5500.329,E2 -5500.329} C_VEL
LIN {X 0,Y 509.873,Z 662.854,A -85,B 0,C 180,E1 -5502.134,E2 -5502.134} C_VEL
LIN {X 0,Y 510.234,Z 653.487,A -85,B 0,C 180,E1 -5503.745,E2 -5503.745} C_VEL
LIN {X 0,Y 510.699,Z 643.853,A -85,B 0,C 180,E1 -5505.157,E2 -5505.157} C_VEL
LIN {X 0,Y 511.213,Z 632.628,A -85,B 0,C 180,E1 -5506.575,E2 -5506.575} C_VEL
LIN {X 0,Y 511.924,Z 620.401,A -85,B 0,C 180,E1 -5507.889,E2 -5507.889} C_VEL
LIN {X 0,Y 512.584,Z 607.807,A -85,B 0,C 180,E1 -5509.041,E2 -5509.041} C_VEL
LIN {X 0,Y 513.334,Z 593.951,A -85,B 0,C 180,E1 -5510.12,E2 -5510.12} C_VEL
LIN {X 0,Y 513.987,Z 580.079,A -85,B 0,C 180,E1 -5511.034,E2 -5511.034} C_VEL
LIN {X 0,Y 514.809,Z 563.907,A -85,B 0,C 180,E1 -5511.901,E2 -5511.901} C_VEL
LIN {X 0,Y 515.398,Z 548.577,A -85,B 0,C 180,E1 -5512.551,E2 -5512.551} C_VEL
LIN {X 0,Y 515.917,Z 532.162,A -85,B 0,C 180,E1 -5513.083,E2 -5513.083} C_VEL
LIN {X 0,Y 516.298,Z 516.812,A -85,B 0,C 180,E1 -5513.436,E2 -5513.436} C_VEL
LIN {X 0,Y 518.098,Z 330.99,A -85,B 0,C 180,E1 -5516.146,E2 -5516.146} C_VEL
LIN {X 0,Y 517.828,Z 326.33,A -85,B 0,C 180,E1 -5516.231,E2 -5516.231} C_VEL
LIN {X 0,Y 514.918,Z 310.413,A -85,B 0,C 180,E1 -5516.645,E2 -5516.645} C_VEL
LIN {X 0,Y 515.735,Z 291.383,A -85,B 0,C 180,E1 -5518.486,E2 -5518.486} C_VEL
LIN {X 0,Y 511.769,Z 277.72,A -85,B 0,C 180,E1 -5520.099,E2 -5520.099} C_VEL
LIN {X 0,Y 509.87,Z 271.288,A -85,B 0,C 180,E1 -5520.889,E2 -5520.889} C_VEL
LIN {X 0,Y 509.857,Z 271.285,A -85,B 0,C 180,E1 -5523.461,E2 -5523.461} C_VEL
LIN {X 0,Y 509.822,Z 271.289,A -85,B 0,C 180,E1 -5526.353,E2 -5526.353} C_VEL
LIN {X 0,Y 509.845,Z 271.291,A -85,B 0,C 180,E1 -5529.352,E2 -5529.352} C_VEL
LIN {X 0,Y 509.846,Z 271.285,A -85,B 0,C 180,E1 -5532.488,E2 -5532.488} C_VEL
LIN {X 0,Y 509.854,Z 271.29,A -85,B 0,C 180,E1 -5535.332,E2 -5535.332} C_VEL
LIN {X 0,Y 509.856,Z 271.282,A -85,B 0,C 180,E1 -5538.575,E2 -5538.575} C_VEL
LIN {X 0,Y 509.848,Z 271.284,A -85,B 0,C 180,E1 -5541.786,E2 -5541.786} C_VEL
LIN {X 0,Y 509.84,Z 271.285,A -85,B 0,C 180,E1 -5544.623,E2 -5544.623} C_VEL
LIN {X 0,Y 509.858,Z 271.287,A -85,B 0,C 180,E1 -5547.481,E2 -5547.481} C_VEL
LIN {X 0,Y 509.855,Z 271.282,A -85,B 0,C 180,E1 -5550.274,E2 -5550.274} C_VEL
LIN {X 0,Y 509.881,Z 271.285,A -85,B 0,C 180,E1 -5552.944,E2 -5552.944} C_VEL
LIN {X 0,Y 509.867,Z 271.285,A -85,B 0,C 180,E1 -5555.574,E2 -5555.574} C_VEL
LIN {X 0,Y 509.847,Z 271.285,A -85,B 0,C 180,E1 -5558.998,E2 -5558.998} C_VEL
LIN {X 0,Y 509.879,Z 271.279,A -85,B 0,C 180,E1 -5562.002,E2 -5562.002} C_VEL
LIN {X 0,Y 509.908,Z 271.281,A -85,B 0,C 180,E1 -5564.819,E2 -5564.819} C_VEL
LIN {X 0,Y 509.898,Z 271.274,A -85,B 0,C 180,E1 -5568.124,E2 -5568.124} C_VEL
LIN {X 0,Y 509.912,Z 271.278,A -85,B 0,C 180,E1 -5571.28,E2 -5571.28} C_VEL
LIN {X 0,Y 509.98,Z 271.26,A -85,B 0,C 180,E1 -5573.671,E2 -5573.671} C_VEL
LIN {X 0,Y 510.054,Z 271.26,A -85,B 0,C 180,E1 -5577.631,E2 -5577.631} C_VEL
LIN {X 0,Y 510.061,Z 271.252,A -85,B 0,C 180,E1 -5580.79,E2 -5580.79} C_VEL
LIN {X 0,Y 509.953,Z 271.277,A -85,B 0,C 180,E1 -5583.16,E2 -5583.16} C_VEL
LIN {X 0,Y 509.951,Z 271.27,A -85,B 0,C 180,E1 -5586.33,E2 -5586.33} C_VEL
LIN {X 0,Y 509.912,Z 271.268,A -85,B 0,C 180,E1 -5588.72,E2 -5588.72} C_VEL
LIN {X 0,Y 509.902,Z 271.278,A -85,B 0,C 180,E1 -5591.932,E2 -5591.932} C_VEL
LIN {X 0,Y 509.892,Z 271.274,A -85,B 0,C 180,E1 -5595.242,E2 -5595.242} C_VEL
LIN {X 0,Y 509.886,Z 271.279,A -85,B 0,C 180,E1 -5598.001,E2 -5598.001} C_VEL
LIN {X 0,Y 509.848,Z 271.281,A -85,B 0,C 180,E1 -5601.002,E2 -5601.002} C_VEL
LIN {X 0,Y 509.868,Z 271.283,A -85,B 0,C 180,E1 -5604.426,E2 -5604.426} C_VEL
LIN {X 0,Y 509.881,Z 271.277,A -85,B 0,C 180,E1 -5607.056,E2 -5607.056} C_VEL
LIN {X 0,Y 509.855,Z 271.283,A -85,B 0,C 180,E1 -5609.751,E2 -5609.751} C_VEL
LIN {X 0,Y 509.871,Z 271.287,A -85,B 0,C 180,E1 -5612.774,E2 -5612.774} C_VEL
LIN {X 0,Y 509.841,Z 271.285,A -85,B 0,C 180,E1 -5615.581,E2 -5615.581} C_VEL
LIN {X 0,Y 509.848,Z 271.279,A -85,B 0,C 180,E1 -5618.338,E2 -5618.338} C_VEL
LIN {X 0,Y 509.855,Z 271.28,A -85,B 0,C 180,E1 -5621.426,E2 -5621.426} C_VEL
LIN {X 0,Y 509.856,Z 271.29,A -85,B 0,C 180,E1 -5624.668,E2 -5624.668} C_VEL
LIN {X 0,Y 509.858,Z 271.285,A -85,B 0,C 180,E1 -5628.103,E2 -5628.103} C_VEL
LIN {X 0,Y 509.847,Z 271.292,A -85,B 0,C 180,E1 -5630.648,E2 -5630.648} C_VEL
LIN {X 0,Y 509.819,Z 271.286,A -85,B 0,C 180,E1 -5633.73,E2 -5633.73} C_VEL
LIN {X 0,Y 509.151,Z 271.374,A -85,B 0,C 180,E1 -5634.39,E2 -5634.39} C_VEL
LIN {X 0,Y 506.34,Z 271.723,A -85,B 0,C 180,E1 -5635.462,E2 -5635.462} C_VEL
LIN {X 0,Y 503.953,Z 272.017,A -85,B 0,C 180,E1 -5636.326,E2 -5636.326} C_VEL
LIN {X 0,Y 502.906,Z 272.144,A -85,B 0,C 180,E1 -5636.992,E2 -5636.992} C_VEL
LIN {X 0,Y 502.808,Z 272.157,A -85,B 0,C 180,E1 -5637.218,E2 -5637.218} C_VEL
LIN {X 0,Y 502.815,Z 272.166,A -85,B 0,C 180,E1 -5640.065,E2 -5640.065} C_VEL
LIN {X 0,Y 502.862,Z 272.334,A -85,B 0,C 180,E1 -5641.288,E2 -5641.288} C_VEL
LIN {X 0,Y 506.44,Z 284.793,A -85,B 0,C 180,E1 -5642.947,E2 -5642.947} C_VEL
LIN {X 0,Y 510.37,Z 293.685,A -85,B 0,C 180,E1 -5643.312,E2 -5643.312} C_VEL
LIN {X 0,Y 511.875,Z 300.957,A -85,B 0,C 180,E1 -5643.51,E2 -5643.51} C_VEL
LIN {X 0,Y 510.003,Z 486.842,A -85,B 0,C 180,E1 -5646.257,E2 -5646.257} C_VEL
LIN {X 0,Y 509.658,Z 502.205,A -85,B 0,C 180,E1 -5646.59,E2 -5646.59} C_VEL
LIN {X 0,Y 509.116,Z 518.589,A -85,B 0,C 180,E1 -5647.101,E2 -5647.101} C_VEL
LIN {X 0,Y 508.485,Z 534.379,A -85,B 0,C 180,E1 -5647.768,E2 -5647.768} C_VEL
LIN {X 0,Y 507.701,Z 549.764,A -85,B 0,C 180,E1 -5648.586,E2 -5648.586} C_VEL
LIN {X 0,Y 506.949,Z 563.984,A -85,B 0,C 180,E1 -5649.51,E2 -5649.51} C_VEL
LIN {X 0,Y 506.205,Z 577.295,A -85,B 0,C 180,E1 -5650.536,E2 -5650.536} C_VEL
LIN {X 0,Y 505.374,Z 590.681,A -85,B 0,C 180,E1 -5651.766,E2 -5651.766} C_VEL
LIN {X 0,Y 504.659,Z 602.069,A -85,B 0,C 180,E1 -5652.995,E2 -5652.995} C_VEL
LIN {X 0,Y 503.969,Z 613.86,A -85,B 0,C 180,E1 -5654.481,E2 -5654.481} C_VEL
LIN {X 0,Y 503.448,Z 623.249,A -85,B 0,C 180,E1 -5655.86,E2 -5655.86} C_VEL
LIN {X 0,Y 502.978,Z 632.626,A -85,B 0,C 180,E1 -5657.492,E2 -5657.492} C_VEL
LIN {X 0,Y 502.655,Z 640.48,A -85,B 0,C 180,E1 -5659.12,E2 -5659.12} C_VEL
LIN {X 0,Y 502.372,Z 647.036,A -85,B 0,C 180,E1 -5660.742,E2 -5660.742} C_VEL
LIN {X 0,Y 502.272,Z 652.331,A -85,B 0,C 180,E1 -5662.361,E2 -5662.361} C_VEL
LIN {X 0,Y 502.189,Z 655.609,A -85,B 0,C 180,E1 -5663.572,E2 -5663.572} C_VEL
LIN {X 0,Y 502.068,Z 658.988,A -85,B 0,C 180,E1 -5665.182,E2 -5665.182} C_VEL
LIN {X 0,Y 502.105,Z 661.44,A -85,B 0,C 180,E1 -5666.79,E2 -5666.79} C_VEL
LIN {X 0,Y 502.032,Z 662.841,A -85,B 0,C 180,E1 -5668.396,E2 -5668.396} C_VEL
LIN {X 0,Y 501.977,Z 663.384,A -85,B 0,C 180,E1 -5670,E2 -5670} C_VEL
LIN {X 0,Y 502.031,Z 662.895,A -85,B 0,C 180,E1 -5671.604,E2 -5671.604} C_VEL
LIN {X 0,Y 502.105,Z 661.547,A -85,B 0,C 180,E1 -5673.21,E2 -5673.21} C_VEL
LIN {X 0,Y 502.066,Z 659.149,A -85,B 0,C 180,E1 -5674.818,E2 -5674.818} C_VEL
LIN {X 0,Y 502.234,Z 655.603,A -85,B 0,C 180,E1 -5676.518,E2 -5676.518} C_VEL
LIN {X 0,Y 502.316,Z 650.144,A -85,B 0,C 180,E1 -5678.448,E2 -5678.448} C_VEL
LIN {X 0,Y 502.574,Z 642.659,A -85,B 0,C 180,E1 -5680.474,E2 -5680.474} C_VEL
LIN {X 0,Y 502.935,Z 634.173,A -85,B 0,C 180,E1 -5682.304,E2 -5682.304} C_VEL
LIN {X 0,Y 503.356,Z 625.018,A -85,B 0,C 180,E1 -5683.937,E2 -5683.937} C_VEL
LIN {X 0,Y 503.923,Z 614.572,A -85,B 0,C 180,E1 -5685.51,E2 -5685.51} C_VEL
LIN {X 0,Y 504.62,Z 602.835,A -85,B 0,C 180,E1 -5687.006,E2 -5687.006} C_VEL
LIN {X 0,Y 505.328,Z 590.534,A -85,B 0,C 180,E1 -5688.34,E2 -5688.34} C_VEL
LIN {X 0,Y 506.147,Z 578.293,A -85,B 0,C 180,E1 -5689.466,E2 -5689.466} C_VEL
LIN {X 0,Y 506.891,Z 565.193,A -85,B 0,C 180,E1 -5690.493,E2 -5690.493} C_VEL
LIN {X 0,Y 507.663,Z 551.258,A -85,B 0,C 180,E1 -5691.415,E2 -5691.415} C_VEL
LIN {X 0,Y 508.363,Z 536.504,A -85,B 0,C 180,E1 -5692.224,E2 -5692.224} C_VEL
LIN {X 0,Y 509.042,Z 520.773,A -85,B 0,C 180,E1 -5692.902,E2 -5692.902} C_VEL
LIN {X 0,Y 509.572,Z 504.346,A -85,B 0,C 180,E1 -5693.441,E2 -5693.441} C_VEL
LIN {X 0,Y 509.944,Z 488.857,A -85,B 0,C 180,E1 -5693.8,E2 -5693.8} C_VEL
LIN {X 0,Y 511.811,Z 300.889,A -85,B 0,C 180,E1 -5696.585,E2 -5696.585} C_VEL
LIN {X 0,Y 509.975,Z 292.667,A -85,B 0,C 180,E1 -5696.816,E2 -5696.816} C_VEL
LIN {X 0,Y 506.375,Z 284.635,A -85,B 0,C 180,E1 -5697.15,E2 -5697.15} C_VEL
LIN {X 0,Y 502.827,Z 272.165,A -85,B 0,C 180,E1 -5698.829,E2 -5698.829} C_VEL
LIN {X 0,Y 502.782,Z 272.167,A -85,B 0,C 180,E1 -5702.084,E2 -5702.084} C_VEL
LIN {X 0,Y 502.796,Z 272.172,A -85,B 0,C 180,E1 -5704.966,E2 -5704.966} C_VEL
LIN {X 0,Y 502.792,Z 272.165,A -85,B 0,C 180,E1 -5708.486,E2 -5708.486} C_VEL
LIN {X 0,Y 502.818,Z 272.166,A -85,B 0,C 180,E1 -5711.066,E2 -5711.066} C_VEL
LIN {X 0,Y 502.799,Z 272.164,A -85,B 0,C 180,E1 -5714.531,E2 -5714.531} C_VEL
LIN {X 0,Y 502.794,Z 272.163,A -85,B 0,C 180,E1 -5717.86,E2 -5717.86} C_VEL
LIN {X 0,Y 502.799,Z 272.168,A -85,B 0,C 180,E1 -5721.024,E2 -5721.024} C_VEL
LIN {X 0,Y 502.781,Z 272.164,A -85,B 0,C 180,E1 -5724.167,E2 -5724.167} C_VEL
LIN {X 0,Y 502.83,Z 272.16,A -85,B 0,C 180,E1 -5726.993,E2 -5726.993} C_VEL
LIN {X 0,Y 502.812,Z 272.161,A -85,B 0,C 180,E1 -5730.065,E2 -5730.065} C_VEL
LIN {X 0,Y 502.83,Z 272.153,A -85,B 0,C 180,E1 -5732.533,E2 -5732.533} C_VEL
LIN {X 0,Y 502.827,Z 272.164,A -85,B 0,C 180,E1 -5735.298,E2 -5735.298} C_VEL
LIN {X 0,Y 502.778,Z 272.157,A -85,B 0,C 180,E1 -5737.826,E2 -5737.826} C_VEL
LIN {X 0,Y 502.821,Z 272.16,A -85,B 0,C 180,E1 -5740.4,E2 -5740.4} C_VEL
LIN {X 0,Y 502.828,Z 272.16,A -85,B 0,C 180,E1 -5742.931,E2 -5742.931} C_VEL
LIN {X 0,Y 502.842,Z 272.16,A -85,B 0,C 180,E1 -5745.429,E2 -5745.429} C_VEL
LIN {X 0,Y 502.874,Z 272.156,A -85,B 0,C 180,E1 -5748.717,E2 -5748.717} C_VEL
LIN {X 0,Y 502.898,Z 272.147,A -85,B 0,C 180,E1 -5751.967,E2 -5751.967} C_VEL
LIN {X 0,Y 502.939,Z 272.146,A -85,B 0,C 180,E1 -5754.386,E2 -5754.386} C_VEL
LIN {X 0,Y 503.023,Z 272.129,A -85,B 0,C 180,E1 -5757.598,E2 -5757.598} C_VEL
LIN {X 0,Y 503.025,Z 272.134,A -85,B 0,C 180,E1 -5760,E2 -5760} C_VEL
LIN {X 0,Y 503.023,Z 272.134,A -85,B 0,C 180,E1 -5762.402,E2 -5762.402} C_VEL
LIN {X 0,Y 502.939,Z 272.144,A -85,B 0,C 180,E1 -5765.613,E2 -5765.613} C_VEL
LIN {X 0,Y 502.898,Z 272.15,A -85,B 0,C 180,E1 -5768.033,E2 -5768.033} C_VEL
LIN {X 0,Y 502.874,Z 272.153,A -85,B 0,C 180,E1 -5771.283,E2 -5771.283} C_VEL
LIN {X 0,Y 502.842,Z 272.161,A -85,B 0,C 180,E1 -5774.571,E2 -5774.571} C_VEL
LIN {X 0,Y 502.859,Z 272.154,A -85,B 0,C 180,E1 -5777.907,E2 -5777.907} C_VEL
LIN {X 0,Y 502.825,Z 272.164,A -85,B 0,C 180,E1 -5780.536,E2 -5780.536} C_VEL
LIN {X 0,Y 502.791,Z 272.17,A -85,B 0,C 180,E1 -5783.04,E2 -5783.04} C_VEL
LIN {X 0,Y 502.837,Z 272.16,A -85,B 0,C 180,E1 -5785.676,E2 -5785.676} C_VEL
LIN {X 0,Y 502.836,Z 272.161,A -85,B 0,C 180,E1 -5788.373,E2 -5788.373} C_VEL
LIN {X 0,Y 502.79,Z 272.167,A -85,B 0,C 180,E1 -5791.499,E2 -5791.499} C_VEL
LIN {X 0,Y 502.804,Z 272.168,A -85,B 0,C 180,E1 -5794.445,E2 -5794.445} C_VEL
LIN {X 0,Y 502.778,Z 272.171,A -85,B 0,C 180,E1 -5797.178,E2 -5797.178} C_VEL
LIN {X 0,Y 502.785,Z 272.167,A -85,B 0,C 180,E1 -5800.015,E2 -5800.015} C_VEL
LIN {X 0,Y 502.8,Z 272.167,A -85,B 0,C 180,E1 -5802.199,E2 -5802.199} C_VEL
LIN {X 0,Y 502.798,Z 272.165,A -85,B 0,C 180,E1 -5805.468,E2 -5805.468} C_VEL
LIN {X 0,Y 502.827,Z 272.161,A -85,B 0,C 180,E1 -5807.864,E2 -5807.864} C_VEL
LIN {X 0,Y 502.799,Z 272.169,A -85,B 0,C 180,E1 -5811.024,E2 -5811.024} C_VEL
LIN {X 0,Y 502.772,Z 272.17,A -85,B 0,C 180,E1 -5814.169,E2 -5814.169} C_VEL
LIN {X 0,Y 502.83,Z 272.165,A -85,B 0,C 180,E1 -5816.994,E2 -5816.994} C_VEL
LIN {X 0,Y 502.846,Z 272.326,A -85,B 0,C 180,E1 -5818.772,E2 -5818.772} C_VEL
LIN {X 0,Y 508.856,Z 292.292,A -85,B 0,C 180,E1 -5821.206,E2 -5821.206} C_VEL
LIN {X 0,Y 509.066,Z 294.525,A -85,B 0,C 180,E1 -5821.444,E2 -5821.444} C_VEL
LIN {X 0,Y 508.308,Z 310.233,A -85,B 0,C 180,E1 -5822.984,E2 -5822.984} C_VEL
LIN {X 0,Y 511.701,Z 329.892,A -85,B 0,C 180,E1 -5823.489,E2 -5823.489} C_VEL
LIN {X 0,Y 509.798,Z 516.606,A -85,B 0,C 180,E1 -5826.247,E2 -5826.247} C_VEL
LIN {X 0,Y 509.398,Z 531.951,A -85,B 0,C 180,E1 -5826.604,E2 -5826.604} C_VEL
LIN {X 0,Y 508.826,Z 548.367,A -85,B 0,C 180,E1 -5827.141,E2 -5827.141} C_VEL
LIN {X 0,Y 508.139,Z 563.896,A -85,B 0,C 180,E1 -5827.806,E2 -5827.806} C_VEL
LIN {X 0,Y 507.31,Z 580.003,A -85,B 0,C 180,E1 -5828.683,E2 -5828.683} C_VEL
LIN {X 0,Y 506.502,Z 595.176,A -85,B 0,C 180,E1 -5829.703,E2 -5829.703} C_VEL
LIN {X 0,Y 505.668,Z 609.356,A -85,B 0,C 180,E1 -5830.846,E2 -5830.846} C_VEL
LIN {X 0,Y 505.005,Z 621.173,A -85,B 0,C 180,E1 -5831.962,E2 -5831.962} C_VEL
LIN {X 0,Y 504.31,Z 632.419,A -85,B 0,C 180,E1 -5833.192,E2 -5833.192} C_VEL
LIN {X 0,Y 503.717,Z 643.641,A -85,B 0,C 180,E1 -5834.628,E2 -5834.628} C_VEL
LIN {X 0,Y 503.172,Z 654.517,A -85,B 0,C 180,E1 -5836.264,E2 -5836.264} C_VEL
LIN {X 0,Y 502.794,Z 663.662,A -85,B 0,C 180,E1 -5837.897,E2 -5837.897} C_VEL
LIN {X 0,Y 502.494,Z 671.324,A -85,B 0,C 180,E1 -5839.524,E2 -5839.524} C_VEL
LIN {X 0,Y 502.257,Z 679.012,A -85,B 0,C 180,E1 -5841.551,E2 -5841.551} C_VEL
LIN {X 0,Y 502.183,Z 684.864,A -85,B 0,C 180,E1 -5843.572,E2 -5843.572} C_VEL
LIN {X 0,Y 502.061,Z 688.283,A -85,B 0,C 180,E1 -5845.182,E2 -5845.182} C_VEL
LIN {X 0,Y 502.102,Z 690.771,A -85,B 0,C 180,E1 -5846.79,E2 -5846.79} C_VEL
LIN {X 0,Y 502.03,Z 692.172,A -85,B 0,C 180,E1 -5848.396,E2 -5848.396} C_VEL
LIN {X 0,Y 501.975,Z 692.7,A -85,B 0,C 180,E1 -5850,E2 -5850} C_VEL
LIN {X 0,Y 502.03,Z 692.172,A -85,B 0,C 180,E1 -5851.604,E2 -5851.604} C_VEL
LIN {X 0,Y 502.102,Z 690.77,A -85,B 0,C 180,E1 -5853.21,E2 -5853.21} C_VEL
LIN {X 0,Y 502.061,Z 688.282,A -85,B 0,C 180,E1 -5854.818,E2 -5854.818} C_VEL
LIN {X 0,Y 502.183,Z 684.758,A -85,B 0,C 180,E1 -5856.469,E2 -5856.469} C_VEL
LIN {X 0,Y 502.257,Z 679.015,A -85,B 0,C 180,E1 -5858.449,E2 -5858.449} C_VEL
LIN {X 0,Y 502.494,Z 671.324,A -85,B 0,C 180,E1 -5860.476,E2 -5860.476} C_VEL
LIN {X 0,Y 502.841,Z 662.644,A -85,B 0,C 180,E1 -5862.307,E2 -5862.307} C_VEL
LIN {X 0,Y 503.226,Z 653.276,A -85,B 0,C 180,E1 -5863.94,E2 -5863.94} C_VEL
LIN {X 0,Y 503.729,Z 643.642,A -85,B 0,C 180,E1 -5865.372,E2 -5865.372} C_VEL
LIN {X 0,Y 504.309,Z 632.418,A -85,B 0,C 180,E1 -5866.808,E2 -5866.808} C_VEL
LIN {X 0,Y 505.044,Z 620.19,A -85,B 0,C 180,E1 -5868.141,E2 -5868.141} C_VEL
LIN {X 0,Y 505.817,Z 606.86,A -85,B 0,C 180,E1 -5869.371,E2 -5869.371} C_VEL
LIN {X 0,Y 506.589,Z 593.741,A -85,B 0,C 180,E1 -5870.399,E2 -5870.399} C_VEL
LIN {X 0,Y 507.3,Z 580.035,A -85,B 0,C 180,E1 -5871.315,E2 -5871.315} C_VEL
LIN {X 0,Y 508.104,Z 565.282,A -85,B 0,C 180,E1 -5872.121,E2 -5872.121} C_VEL
LIN {X 0,Y 508.768,Z 549.671,A -85,B 0,C 180,E1 -5872.808,E2 -5872.808} C_VEL
LIN {X 0,Y 509.356,Z 532.872,A -85,B 0,C 180,E1 -5873.371,E2 -5873.371} C_VEL
LIN {X 0,Y 509.797,Z 516.605,A -85,B 0,C 180,E1 -5873.754,E2 -5873.754} C_VEL
LIN {X 0,Y 511.713,Z 330.779,A -85,B 0,C 180,E1 -5876.497,E2 -5876.497} C_VEL
LIN {X 0,Y 511.303,Z 326.738,A -85,B 0,C 180,E1 -5876.582,E2 -5876.582} C_VEL
LIN {X 0,Y 508.295,Z 310.287,A -85,B 0,C 180,E1 -5877.011,E2 -5877.011} C_VEL
LIN {X 0,Y 509.108,Z 293.404,A -85,B 0,C 180,E1 -5878.666,E2 -5878.666} C_VEL
LIN {X 0,Y 503.93,Z 275.76,A -85,B 0,C 180,E1 -5880.796,E2 -5880.796} C_VEL
LIN {X 0,Y 502.815,Z 272.168,A -85,B 0,C 180,E1 -5881.275,E2 -5881.275} C_VEL
LIN {X 0,Y 502.801,Z 272.166,A -85,B 0,C 180,E1 -5883.994,E2 -5883.994} C_VEL
LIN {X 0,Y 502.775,Z 272.173,A -85,B 0,C 180,E1 -5887.178,E2 -5887.178} C_VEL
LIN {X 0,Y 502.786,Z 272.167,A -85,B 0,C 180,E1 -5890.015,E2 -5890.015} C_VEL
LIN {X 0,Y 502.801,Z 272.163,A -85,B 0,C 180,E1 -5892.199,E2 -5892.199} C_VEL
LIN {X 0,Y 502.798,Z 272.166,A -85,B 0,C 180,E1 -5895.468,E2 -5895.468} C_VEL
LIN {X 0,Y 502.818,Z 272.162,A -85,B 0,C 180,E1 -5898.934,E2 -5898.934} C_VEL
LIN {X 0,Y 502.791,Z 272.161,A -85,B 0,C 180,E1 -5902.046,E2 -5902.046} C_VEL
LIN {X 0,Y 502.805,Z 272.165,A -85,B 0,C 180,E1 -5905.035,E2 -5905.035} C_VEL
LIN {X 0,Y 502.78,Z 272.165,A -85,B 0,C 180,E1 -5907.915,E2 -5907.915} C_VEL
LIN {X 0,Y 502.821,Z 272.16,A -85,B 0,C 180,E1 -5910.712,E2 -5910.712} C_VEL
LIN {X 0,Y 502.86,Z 272.16,A -85,B 0,C 180,E1 -5913.439,E2 -5913.439} C_VEL
LIN {X 0,Y 502.789,Z 272.163,A -85,B 0,C 180,E1 -5916.086,E2 -5916.086} C_VEL
LIN {X 0,Y 502.78,Z 272.166,A -85,B 0,C 180,E1 -5918.689,E2 -5918.689} C_VEL
LIN {X 0,Y 502.826,Z 272.16,A -85,B 0,C 180,E1 -5921.248,E2 -5921.248} C_VEL
LIN {X 0,Y 502.819,Z 272.16,A -85,B 0,C 180,E1 -5923.767,E2 -5923.767} C_VEL
LIN {X 0,Y 502.828,Z 272.149,A -85,B 0,C 180,E1 -5926.255,E2 -5926.255} C_VEL
LIN {X 0,Y 502.875,Z 272.153,A -85,B 0,C 180,E1 -5928.717,E2 -5928.717} C_VEL
LIN {X 0,Y 502.899,Z 272.145,A -85,B 0,C 180,E1 -5931.967,E2 -5931.967} C_VEL
LIN {X 0,Y 502.939,Z 272.136,A -85,B 0,C 180,E1 -5934.387,E2 -5934.387} C_VEL
LIN {X 0,Y 503.023,Z 272.136,A -85,B 0,C 180,E1 -5937.598,E2 -5937.598} C_VEL
LIN {X 0,Y 503.025,Z 272.125,A -85,B 0,C 180,E1 -5940,E2 -5940} C_VEL
LIN {X 0,Y 503.023,Z 272.129,A -85,B 0,C 180,E1 -5942.402,E2 -5942.402} C_VEL
LIN {X 0,Y 502.931,Z 272.145,A -85,B 0,C 180,E1 -5945.614,E2 -5945.614} C_VEL
LIN {X 0,Y 502.899,Z 272.137,A -85,B 0,C 180,E1 -5948.033,E2 -5948.033} C_VEL
LIN {X 0,Y 502.875,Z 272.158,A -85,B 0,C 180,E1 -5951.283,E2 -5951.283} C_VEL
LIN {X 0,Y 502.843,Z 272.155,A -85,B 0,C 180,E1 -5954.571,E2 -5954.571} C_VEL
LIN {X 0,Y 502.86,Z 272.154,A -85,B 0,C 180,E1 -5957.907,E2 -5957.907} C_VEL
LIN {X 0,Y 502.827,Z 272.16,A -85,B 0,C 180,E1 -5960.536,E2 -5960.536} C_VEL
LIN {X 0,Y 502.792,Z 272.163,A -85,B 0,C 180,E1 -5963.041,E2 -5963.041} C_VEL
LIN {X 0,Y 502.838,Z 272.157,A -85,B 0,C 180,E1 -5965.676,E2 -5965.676} C_VEL
LIN {X 0,Y 502.838,Z 272.15,A -85,B 0,C 180,E1 -5968.373,E2 -5968.373} C_VEL
LIN {X 0,Y 502.791,Z 272.163,A -85,B 0,C 180,E1 -5971.499,E2 -5971.499} C_VEL
LIN {X 0,Y 502.805,Z 272.164,A -85,B 0,C 180,E1 -5974.445,E2 -5974.445} C_VEL
LIN {X 0,Y 502.779,Z 272.162,A -85,B 0,C 180,E1 -5977.179,E2 -5977.179} C_VEL
LIN {X 0,Y 502.786,Z 272.163,A -85,B 0,C 180,E1 -5980.015,E2 -5980.015} C_VEL
LIN {X 0,Y 502.801,Z 272.158,A -85,B 0,C 180,E1 -5982.199,E2 -5982.199} C_VEL
LIN {X 0,Y 502.8,Z 272.159,A -85,B 0,C 180,E1 -5985.468,E2 -5985.468} C_VEL
LIN {X 0,Y 502.82,Z 272.167,A -85,B 0,C 180,E1 -5988.934,E2 -5988.934} C_VEL
LIN {X 0,Y 502.793,Z 272.161,A -85,B 0,C 180,E1 -5992.046,E2 -5992.046} C_VEL
LIN {X 0,Y 502.798,Z 272.168,A -85,B 0,C 180,E1 -5995.034,E2 -5995.034} C_VEL
LIN {X 0,Y 502.808,Z 272.157,A -85,B 0,C 180,E1 -5997.218,E2 -5997.218} C_VEL
LIN {X 0,Y 502.096,Z 272.251,A -85,B 0,C 180,E1 -5997.886,E2 -5997.886} C_VEL
LIN {X 0,Y 499.203,Z 272.616,A -85,B 0,C 180,E1 -5998.972,E2 -5998.972} C_VEL
LIN {X 0,Y 496.814,Z 272.914,A -85,B 0,C 180,E1 -5999.847,E2 -5999.847} C_VEL
LIN {X 0,Y 495.839,Z 273.035,A -85,B 0,C 180,E1 -6000.523,E2 -6000.523} C_VEL
LIN {X 0,Y 495.785,Z 273.041,A -85,B 0,C 180,E1 -6000.751,E2 -6000.751} C_VEL
LIN {X 0,Y 495.83,Z 273.266,A -85,B 0,C 180,E1 -6000.928,E2 -6000.928} C_VEL
LIN {X 0,Y 499.281,Z 284.991,A -85,B 0,C 180,E1 -6002.526,E2 -6002.526} C_VEL
LIN {X 0,Y 504.404,Z 296.674,A -85,B 0,C 180,E1 -6003.014,E2 -6003.014} C_VEL
LIN {X 0,Y 505.562,Z 302.835,A -85,B 0,C 180,E1 -6003.178,E2 -6003.178} C_VEL
LIN {X 0,Y 503.538,Z 487.083,A -85,B 0,C 180,E1 -6005.933,E2 -6005.933} C_VEL
LIN {X 0,Y 503.142,Z 502.435,A -85,B 0,C 180,E1 -6006.268,E2 -6006.268} C_VEL
LIN {X 0,Y 502.582,Z 518.813,A -85,B 0,C 180,E1 -6006.786,E2 -6006.786} C_VEL
LIN {X 0,Y 501.884,Z 535.267,A -85,B 0,C 180,E1 -6007.492,E2 -6007.492} C_VEL
LIN {X 0,Y 501.101,Z 549.983,A -85,B 0,C 180,E1 -6008.29,E2 -6008.29} C_VEL
LIN {X 0,Y 500.275,Z 564.202,A -85,B 0,C 180,E1 -6009.224,E2 -6009.224} C_VEL
LIN {X 0,Y 499.45,Z 577.512,A -85,B 0,C 180,E1 -6010.262,E2 -6010.262} C_VEL
LIN {X 0,Y 498.584,Z 590.896,A -85,B 0,C 180,E1 -6011.509,E2 -6011.509} C_VEL
LIN {X 0,Y 497.822,Z 602.284,A -85,B 0,C 180,E1 -6012.755,E2 -6012.755} C_VEL
LIN {X 0,Y 497.088,Z 613.456,A -85,B 0,C 180,E1 -6014.173,E2 -6014.173} C_VEL
LIN {X 0,Y 496.514,Z 623.462,A -85,B 0,C 180,E1 -6015.658,E2 -6015.658} C_VEL
LIN {X 0,Y 495.966,Z 632.84,A -85,B 0,C 180,E1 -6017.312,E2 -6017.312} C_VEL
LIN {X 0,Y 495.628,Z 640.692,A -85,B 0,C 180,E1 -6018.964,E2 -6018.964} C_VEL
LIN {X 0,Y 495.32,Z 647.246,A -85,B 0,C 180,E1 -6020.609,E2 -6020.609} C_VEL
LIN {X 0,Y 495.212,Z 652.541,A -85,B 0,C 180,E1 -6022.252,E2 -6022.252} C_VEL
LIN {X 0,Y 495.127,Z 655.912,A -85,B 0,C 180,E1 -6023.516,E2 -6023.516} C_VEL
LIN {X 0,Y 494.994,Z 659.196,A -85,B 0,C 180,E1 -6025.113,E2 -6025.113} C_VEL
LIN {X 0,Y 495.026,Z 661.648,A -85,B 0,C 180,E1 -6026.744,E2 -6026.744} C_VEL
LIN {X 0,Y 494.959,Z 663.048,A -85,B 0,C 180,E1 -6028.373,E2 -6028.373} C_VEL
LIN {X 0,Y 494.895,Z 663.591,A -85,B 0,C 180,E1 -6030,E2 -6030} C_VEL
LIN {X 0,Y 494.958,Z 663.101,A -85,B 0,C 180,E1 -6031.627,E2 -6031.627} C_VEL
LIN {X 0,Y 495.026,Z 661.753,A -85,B 0,C 180,E1 -6033.255,E2 -6033.255} C_VEL
LIN {X 0,Y 494.992,Z 659.355,A -85,B 0,C 180,E1 -6034.887,E2 -6034.887} C_VEL
LIN {X 0,Y 495.13,Z 656.041,A -85,B 0,C 180,E1 -6036.52,E2 -6036.52} C_VEL
LIN {X 0,Y 495.274,Z 650.35,A -85,B 0,C 180,E1 -6038.569,E2 -6038.569} C_VEL
LIN {X 0,Y 495.555,Z 642.865,A -85,B 0,C 180,E1 -6040.624,E2 -6040.624} C_VEL
LIN {X 0,Y 495.922,Z 634.38,A -85,B 0,C 180,E1 -6042.481,E2 -6042.481} C_VEL
LIN {X 0,Y 496.413,Z 625.223,A -85,B 0,C 180,E1 -6044.135,E2 -6044.135} C_VEL
LIN {X 0,Y 496.974,Z 615.799,A -85,B 0,C 180,E1 -6045.586,E2 -6045.586} C_VEL
LIN {X 0,Y 497.665,Z 604.808,A -85,B 0,C 180,E1 -6047.039,E2 -6047.039} C_VEL
LIN {X 0,Y 498.479,Z 591.793,A -85,B 0,C 180,E1 -6048.495,E2 -6048.495} C_VEL
LIN {X 0,Y 499.319,Z 579.593,A -85,B 0,C 180,E1 -6049.642,E2 -6049.642} C_VEL
LIN {X 0,Y 500.222,Z 565.392,A -85,B 0,C 180,E1 -6050.778,E2 -6050.778} C_VEL
LIN {X 0,Y 501.02,Z 551.604,A -85,B 0,C 180,E1 -6051.704,E2 -6051.704} C_VEL
LIN {X 0,Y 501.763,Z 537.101,A -85,B 0,C 180,E1 -6052.51,E2 -6052.51} C_VEL
LIN {X 0,Y 502.448,Z 522.261,A -85,B 0,C 180,E1 -6053.166,E2 -6053.166} C_VEL
LIN {X 0,Y 503.06,Z 505.445,A -85,B 0,C 180,E1 -6053.736,E2 -6053.736} C_VEL
LIN {X 0,Y 503.481,Z 490.531,A -85,B 0,C 180,E1 -6054.098,E2 -6054.098} C_VEL
LIN {X 0,Y 505.485,Z 301.98,A -85,B 0,C 180,E1 -6056.93,E2 -6056.93} C_VEL
LIN {X 0,Y 504.014,Z 295.496,A -85,B 0,C 180,E1 -6057.118,E2 -6057.118} C_VEL
LIN {X 0,Y 499.176,Z 284.763,A -85,B 0,C 180,E1 -6057.585,E2 -6057.585} C_VEL
LIN {X 0,Y 495.779,Z 273.037,A -85,B 0,C 180,E1 -6059.22,E2 -6059.22} C_VEL
LIN {X 0,Y 495.767,Z 273.036,A -85,B 0,C 180,E1 -6062.594,E2 -6062.594} C_VEL
LIN {X 0,Y 495.744,Z 273.04,A -85,B 0,C 180,E1 -6065.538,E2 -6065.538} C_VEL
LIN {X 0,Y 495.761,Z 273.043,A -85,B 0,C 180,E1 -6068.768,E2 -6068.768} C_VEL
LIN {X 0,Y 495.755,Z 273.04,A -85,B 0,C 180,E1 -6071.781,E2 -6071.781} C_VEL
LIN {X 0,Y 495.748,Z 273.044,A -85,B 0,C 180,E1 -6075.139,E2 -6075.139} C_VEL
LIN {X 0,Y 495.755,Z 273.039,A -85,B 0,C 180,E1 -6078.219,E2 -6078.219} C_VEL
LIN {X 0,Y 495.748,Z 273.045,A -85,B 0,C 180,E1 -6081.408,E2 -6081.408} C_VEL
LIN {X 0,Y 495.753,Z 273.04,A -85,B 0,C 180,E1 -6084.463,E2 -6084.463} C_VEL
LIN {X 0,Y 495.765,Z 273.038,A -85,B 0,C 180,E1 -6087.405,E2 -6087.405} C_VEL
LIN {X 0,Y 495.764,Z 273.039,A -85,B 0,C 180,E1 -6090.253,E2 -6090.253} C_VEL
LIN {X 0,Y 495.821,Z 273.033,A -85,B 0,C 180,E1 -6093.251,E2 -6093.251} C_VEL
LIN {X 0,Y 495.75,Z 273.041,A -85,B 0,C 180,E1 -6095.725,E2 -6095.725} C_VEL
LIN {X 0,Y 495.74,Z 273.033,A -85,B 0,C 180,E1 -6098.371,E2 -6098.371} C_VEL
LIN {X 0,Y 495.781,Z 273.043,A -85,B 0,C 180,E1 -6100.971,E2 -6100.971} C_VEL
LIN {X 0,Y 495.775,Z 273.029,A -85,B 0,C 180,E1 -6103.53,E2 -6103.53} C_VEL
LIN {X 0,Y 495.791,Z 273.034,A -85,B 0,C 180,E1 -6106.055,E2 -6106.055} C_VEL
LIN {X 0,Y 495.849,Z 273.03,A -85,B 0,C 180,E1 -6108.555,E2 -6108.555} C_VEL
LIN {X 0,Y 495.869,Z 273.022,A -85,B 0,C 180,E1 -6111.852,E2 -6111.852} C_VEL
LIN {X 0,Y 495.896,Z 273.023,A -85,B 0,C 180,E1 -6114.306,E2 -6114.306} C_VEL
LIN {X 0,Y 495.991,Z 273.005,A -85,B 0,C 180,E1 -6117.564,E2 -6117.564} C_VEL
LIN {X 0,Y 495.996,Z 273.01,A -85,B 0,C 180,E1 -6120,E2 -6120} C_VEL
LIN {X 0,Y 495.991,Z 273.01,A -85,B 0,C 180,E1 -6122.436,E2 -6122.436} C_VEL
LIN {X 0,Y 495.896,Z 273.021,A -85,B 0,C 180,E1 -6125.693,E2 -6125.693} C_VEL
LIN {X 0,Y 495.87,Z 273.026,A -85,B 0,C 180,E1 -6128.148,E2 -6128.148} C_VEL
LIN {X 0,Y 495.849,Z 273.027,A -85,B 0,C 180,E1 -6131.445,E2 -6131.445} C_VEL
LIN {X 0,Y 495.787,Z 273.043,A -85,B 0,C 180,E1 -6134.783,E2 -6134.783} C_VEL
LIN {X 0,Y 495.783,Z 273.039,A -85,B 0,C 180,E1 -6137.319,E2 -6137.319} C_VEL
LIN {X 0,Y 495.768,Z 273.039,A -85,B 0,C 180,E1 -6139.89,E2 -6139.89} C_VEL
LIN {X 0,Y 495.758,Z 273.048,A -85,B 0,C 180,E1 -6142.861,E2 -6142.861} C_VEL
LIN {X 0,Y 495.787,Z 273.038,A -85,B 0,C 180,E1 -6146.068,E2 -6146.068} C_VEL
LIN {X 0,Y 495.769,Z 273.048,A -85,B 0,C 180,E1 -6148.815,E2 -6148.815} C_VEL
LIN {X 0,Y 495.753,Z 273.043,A -85,B 0,C 180,E1 -6151.725,E2 -6151.725} C_VEL
LIN {X 0,Y 495.774,Z 273.048,A -85,B 0,C 180,E1 -6154.695,E2 -6154.695} C_VEL
LIN {X 0,Y 495.728,Z 273.047,A -85,B 0,C 180,E1 -6157.562,E2 -6157.562} C_VEL
LIN {X 0,Y 495.764,Z 273.049,A -85,B 0,C 180,E1 -6160.7,E2 -6160.7} C_VEL
LIN {X 0,Y 495.731,Z 273.046,A -85,B 0,C 180,E1 -6164.001,E2 -6164.001} C_VEL
LIN {X 0,Y 495.731,Z 273.049,A -85,B 0,C 180,E1 -6167.118,E2 -6167.118} C_VEL
LIN {X 0,Y 495.756,Z 273.042,A -85,B 0,C 180,E1 -6169.953,E2 -6169.953} C_VEL
LIN {X 0,Y 495.725,Z 273.051,A -85,B 0,C 180,E1 -6172.553,E2 -6172.553} C_VEL
LIN {X 0,Y 495.775,Z 273.031,A -85,B 0,C 180,E1 -6175.457,E2 -6175.457} C_VEL
LIN {X 0,Y 495.782,Z 273.181,A -85,B 0,C 180,E1 -6178.39,E2 -6178.39} C_VEL
LIN {X 0,Y 501.845,Z 293.192,A -85,B 0,C 180,E1 -6180.88,E2 -6180.88} C_VEL
LIN {X 0,Y 502.454,Z 295.433,A -85,B 0,C 180,E1 -6181.147,E2 -6181.147} C_VEL
LIN {X 0,Y 501.691,Z 310.046,A -85,B 0,C 180,E1 -6182.6,E2 -6182.6} C_VEL
LIN {X 0,Y 505.338,Z 330.798,A -85,B 0,C 180,E1 -6183.145,E2 -6183.145} C_VEL
LIN {X 0,Y 503.313,Z 516.4,A -85,B 0,C 180,E1 -6185.921,E2 -6185.921} C_VEL
LIN {X 0,Y 502.872,Z 531.743,A -85,B 0,C 180,E1 -6186.282,E2 -6186.282} C_VEL
LIN {X 0,Y 502.33,Z 546.855,A -85,B 0,C 180,E1 -6186.774,E2 -6186.774} C_VEL
LIN {X 0,Y 501.606,Z 562.353,A -85,B 0,C 180,E1 -6187.435,E2 -6187.435} C_VEL
LIN {X 0,Y 500.822,Z 576.851,A -85,B 0,C 180,E1 -6188.213,E2 -6188.213} C_VEL
LIN {X 0,Y 500.016,Z 590.667,A -85,B 0,C 180,E1 -6189.105,E2 -6189.105} C_VEL
LIN {X 0,Y 499.135,Z 605.445,A -85,B 0,C 180,E1 -6190.249,E2 -6190.249} C_VEL
LIN {X 0,Y 498.221,Z 618.946,A -85,B 0,C 180,E1 -6191.495,E2 -6191.495} C_VEL
LIN {X 0,Y 497.503,Z 630.415,A -85,B 0,C 180,E1 -6192.743,E2 -6192.743} C_VEL
LIN {X 0,Y 496.827,Z 641.478,A -85,B 0,C 180,E1 -6194.135,E2 -6194.135} C_VEL
LIN {X 0,Y 496.262,Z 651.819,A -85,B 0,C 180,E1 -6195.651,E2 -6195.651} C_VEL
LIN {X 0,Y 495.846,Z 661.329,A -85,B 0,C 180,E1 -6197.309,E2 -6197.309} C_VEL
LIN {X 0,Y 495.508,Z 669.289,A -85,B 0,C 180,E1 -6198.961,E2 -6198.961} C_VEL
LIN {X 0,Y 495.23,Z 675.932,A -85,B 0,C 180,E1 -6200.607,E2 -6200.607} C_VEL
LIN {X 0,Y 495.138,Z 681.324,A -85,B 0,C 180,E1 -6202.251,E2 -6202.251} C_VEL
LIN {X 0,Y 495.084,Z 684.848,A -85,B 0,C 180,E1 -6203.558,E2 -6203.558} C_VEL
LIN {X 0,Y 494.983,Z 688.075,A -85,B 0,C 180,E1 -6205.113,E2 -6205.113} C_VEL
LIN {X 0,Y 495.022,Z 690.564,A -85,B 0,C 180,E1 -6206.745,E2 -6206.745} C_VEL
LIN {X 0,Y 494.955,Z 691.966,A -85,B 0,C 180,E1 -6208.373,E2 -6208.373} C_VEL
LIN {X 0,Y 494.893,Z 692.493,A -85,B 0,C 180,E1 -6210,E2 -6210} C_VEL
LIN {X 0,Y 494.955,Z 691.965,A -85,B 0,C 180,E1 -6211.627,E2 -6211.627} C_VEL
LIN {X 0,Y 495.022,Z 690.563,A -85,B 0,C 180,E1 -6213.256,E2 -6213.256} C_VEL
LIN {X 0,Y 494.983,Z 688.075,A -85,B 0,C 180,E1 -6214.887,E2 -6214.887} C_VEL
LIN {X 0,Y 495.085,Z 684.658,A -85,B 0,C 180,E1 -6216.521,E2 -6216.521} C_VEL
LIN {X 0,Y 495.174,Z 680.073,A -85,B 0,C 180,E1 -6218.159,E2 -6218.159} C_VEL
LIN {X 0,Y 495.259,Z 674.391,A -85,B 0,C 180,E1 -6219.804,E2 -6219.804} C_VEL
LIN {X 0,Y 495.63,Z 667.465,A -85,B 0,C 180,E1 -6221.45,E2 -6221.45} C_VEL
LIN {X 0,Y 495.919,Z 659.076,A -85,B 0,C 180,E1 -6223.106,E2 -6223.106} C_VEL
LIN {X 0,Y 496.482,Z 649.109,A -85,B 0,C 180,E1 -6224.762,E2 -6224.762} C_VEL
LIN {X 0,Y 497.042,Z 638.774,A -85,B 0,C 180,E1 -6226.227,E2 -6226.227} C_VEL
LIN {X 0,Y 497.753,Z 626.824,A -85,B 0,C 180,E1 -6227.672,E2 -6227.672} C_VEL
LIN {X 0,Y 498.558,Z 614.647,A -85,B 0,C 180,E1 -6228.918,E2 -6228.918} C_VEL
LIN {X 0,Y 499.31,Z 601.629,A -85,B 0,C 180,E1 -6230.065,E2 -6230.065} C_VEL
LIN {X 0,Y 500.167,Z 587.692,A -85,B 0,C 180,E1 -6231.104,E2 -6231.104} C_VEL
LIN {X 0,Y 501.092,Z 572.694,A -85,B 0,C 180,E1 -6232.028,E2 -6232.028} C_VEL
LIN {X 0,Y 501.801,Z 557.49,A -85,B 0,C 180,E1 -6232.789,E2 -6232.789} C_VEL
LIN {X 0,Y 502.566,Z 540.958,A -85,B 0,C 180,E1 -6233.433,E2 -6233.433} C_VEL
LIN {X 0,Y 503.085,Z 524.815,A -85,B 0,C 180,E1 -6233.899,E2 -6233.899} C_VEL
LIN {X 0,Y 503.49,Z 508.818,A -85,B 0,C 180,E1 -6234.207,E2 -6234.207} C_VEL
LIN {X 0,Y 505.341,Z 330.407,A -85,B 0,C 180,E1 -6236.86,E2 -6236.86} C_VEL
LIN {X 0,Y 501.728,Z 310.055,A -85,B 0,C 180,E1 -6237.396,E2 -6237.396} C_VEL
LIN {X 0,Y 502.469,Z 295.419,A -85,B 0,C 180,E1 -6238.852,E2 -6238.852} C_VEL
LIN {X 0,Y 496.566,Z 275.676,A -85,B 0,C 180,E1 -6241.289,E2 -6241.289} C_VEL
LIN {X 0,Y 495.753,Z 273.046,A -85,B 0,C 180,E1 -6241.636,E2 -6241.636} C_VEL
LIN {X 0,Y 495.775,Z 273.041,A -85,B 0,C 180,E1 -6244.543,E2 -6244.543} C_VEL
LIN {X 0,Y 495.727,Z 273.049,A -85,B 0,C 180,E1 -6247.562,E2 -6247.562} C_VEL
LIN {X 0,Y 495.765,Z 273.042,A -85,B 0,C 180,E1 -6250.7,E2 -6250.7} C_VEL
LIN {X 0,Y 495.733,Z 273.045,A -85,B 0,C 180,E1 -6253.695,E2 -6253.695} C_VEL
LIN {X 0,Y 495.725,Z 273.041,A -85,B 0,C 180,E1 -6256.305,E2 -6256.305} C_VEL
LIN {X 0,Y 495.764,Z 273.044,A -85,B 0,C 180,E1 -6259.3,E2 -6259.3} C_VEL
LIN {X 0,Y 495.728,Z 273.041,A -85,B 0,C 180,E1 -6262.438,E2 -6262.438} C_VEL
LIN {X 0,Y 495.781,Z 273.041,A -85,B 0,C 180,E1 -6265.457,E2 -6265.457} C_VEL
LIN {X 0,Y 495.752,Z 273.04,A -85,B 0,C 180,E1 -6268.364,E2 -6268.364} C_VEL
LIN {X 0,Y 495.785,Z 273.04,A -85,B 0,C 180,E1 -6271.507,E2 -6271.507} C_VEL
LIN {X 0,Y 495.788,Z 273.037,A -85,B 0,C 180,E1 -6273.932,E2 -6273.932} C_VEL
LIN {X 0,Y 495.759,Z 273.047,A -85,B 0,C 180,E1 -6277.139,E2 -6277.139} C_VEL
LIN {X 0,Y 495.768,Z 273.027,A -85,B 0,C 180,E1 -6280.11,E2 -6280.11} C_VEL
LIN {X 0,Y 495.779,Z 273.039,A -85,B 0,C 180,E1 -6282.681,E2 -6282.681} C_VEL
LIN {X 0,Y 495.787,Z 273.033,A -85,B 0,C 180,E1 -6285.217,E2 -6285.217} C_VEL
LIN {X 0,Y 495.849,Z 273.026,A -85,B 0,C 180,E1 -6288.555,E2 -6288.555} C_VEL
LIN {X 0,Y 495.87,Z 273.021,A -85,B 0,C 180,E1 -6291.852,E2 -6291.852} C_VEL
LIN {X 0,Y 495.896,Z 273.012,A -85,B 0,C 180,E1 -6294.307,E2 -6294.307} C_VEL
LIN {X 0,Y 495.992,Z 273.012,A -85,B 0,C 180,E1 -6297.564,E2 -6297.564} C_VEL
LIN {X 0,Y 495.981,Z 273.004,A -85,B 0,C 180,E1 -6300.812,E2 -6300.812} C_VEL
LIN {X 0,Y 495.992,Z 273.005,A -85,B 0,C 180,E1 -6302.436,E2 -6302.436} C_VEL
LIN {X 0,Y 495.887,Z 273.022,A -85,B 0,C 180,E1 -6305.694,E2 -6305.694} C_VEL
LIN {X 0,Y 495.871,Z 273.012,A -85,B 0,C 180,E1 -6308.148,E2 -6308.148} C_VEL
LIN {X 0,Y 495.849,Z 273.031,A -85,B 0,C 180,E1 -6311.445,E2 -6311.445} C_VEL
LIN {X 0,Y 495.788,Z 273.031,A -85,B 0,C 180,E1 -6314.783,E2 -6314.783} C_VEL
LIN {X 0,Y 495.785,Z 273.04,A -85,B 0,C 180,E1 -6317.319,E2 -6317.319} C_VEL
LIN {X 0,Y 495.769,Z 273.036,A -85,B 0,C 180,E1 -6319.891,E2 -6319.891} C_VEL
LIN {X 0,Y 495.76,Z 273.035,A -85,B 0,C 180,E1 -6322.861,E2 -6322.861} C_VEL
LIN {X 0,Y 495.789,Z 273.035,A -85,B 0,C 180,E1 -6326.068,E2 -6326.068} C_VEL
LIN {X 0,Y 495.77,Z 273.035,A -85,B 0,C 180,E1 -6328.815,E2 -6328.815} C_VEL
LIN {X 0,Y 495.753,Z 273.038,A -85,B 0,C 180,E1 -6331.725,E2 -6331.725} C_VEL
LIN {X 0,Y 495.775,Z 273.042,A -85,B 0,C 180,E1 -6334.695,E2 -6334.695} C_VEL
LIN {X 0,Y 495.729,Z 273.036,A -85,B 0,C 180,E1 -6337.562,E2 -6337.562} C_VEL
LIN {X 0,Y 495.765,Z 273.044,A -85,B 0,C 180,E1 -6340.7,E2 -6340.7} C_VEL
LIN {X 0,Y 495.733,Z 273.043,A -85,B 0,C 180,E1 -6344.001,E2 -6344.001} C_VEL
LIN {X 0,Y 495.725,Z 273.049,A -85,B 0,C 180,E1 -6347.117,E2 -6347.117} C_VEL
LIN {X 0,Y 495.759,Z 273.04,A -85,B 0,C 180,E1 -6349.953,E2 -6349.953} C_VEL
LIN {X 0,Y 495.727,Z 273.036,A -85,B 0,C 180,E1 -6352.553,E2 -6352.553} C_VEL
LIN {X 0,Y 495.777,Z 273.039,A -85,B 0,C 180,E1 -6355.457,E2 -6355.457} C_VEL
LIN {X 0,Y 495.755,Z 273.045,A -85,B 0,C 180,E1 -6358.364,E2 -6358.364} C_VEL
LIN {X 0,Y 495.785,Z 273.041,A -85,B 0,C 180,E1 -6360.751,E2 -6360.751} C_VEL
LIN {X 0,Y 495.735,Z 273.742,A -85,B 0,C 180,E1 -6360.961,E2 -6360.961} C_VEL
LIN {X 0,Y 495.225,Z 276.881,A -85,B 0,C 180,E1 -6361.319,E2 -6361.319} C_VEL
LIN {X 0,Y 493.864,Z 282.014,A -85,B 0,C 180,E1 -6361.808,E2 -6361.808} C_VEL
LIN {X 0,Y 493.443,Z 286.308,A -85,B 0,C 180,E1 -6362.111,E2 -6362.111} C_VEL
LIN {X 0,Y 494.095,Z 289.637,A -85,B 0,C 180,E1 -6362.284,E2 -6362.284} C_VEL
LIN {X 0,Y 498.465,Z 299.63,A -85,B 0,C 180,E1 -6362.71,E2 -6362.71} C_VEL
LIN {X 0,Y 499.241,Z 304.171,A -85,B 0,C 180,E1 -6362.828,E2 -6362.828} C_VEL
LIN {X 0,Y 497.063,Z 487.319,A -85,B 0,C 180,E1 -6365.599,E2 -6365.599} C_VEL
LIN {X 0,Y 496.653,Z 502.66,A -85,B 0,C 180,E1 -6365.939,E2 -6365.939} C_VEL
LIN {X 0,Y 496.08,Z 519.034,A -85,B 0,C 180,E1 -6366.464,E2 -6366.464} C_VEL
LIN {X 0,Y 495.357,Z 534.65,A -85,B 0,C 180,E1 -6367.138,E2 -6367.138} C_VEL
LIN {X 0,Y 494.601,Z 548.689,A -85,B 0,C 180,E1 -6367.895,E2 -6367.895} C_VEL
LIN {X 0,Y 493.816,Z 561.56,A -85,B 0,C 180,E1 -6368.721,E2 -6368.721} C_VEL
LIN {X 0,Y 492.791,Z 576.478,A -85,B 0,C 180,E1 -6369.876,E2 -6369.876} C_VEL
LIN {X 0,Y 491.83,Z 590.052,A -85,B 0,C 180,E1 -6371.138,E2 -6371.138} C_VEL
LIN {X 0,Y 490.974,Z 602.499,A -85,B 0,C 180,E1 -6372.506,E2 -6372.506} C_VEL
LIN {X 0,Y 490.177,Z 614.135,A -85,B 0,C 180,E1 -6374.011,E2 -6374.011} C_VEL
LIN {X 0,Y 489.587,Z 623.675,A -85,B 0,C 180,E1 -6375.451,E2 -6375.451} C_VEL
LIN {X 0,Y 488.984,Z 633.052,A -85,B 0,C 180,E1 -6377.128,E2 -6377.128} C_VEL
LIN {X 0,Y 488.607,Z 640.904,A -85,B 0,C 180,E1 -6378.803,E2 -6378.803} C_VEL
LIN {X 0,Y 488.279,Z 647.457,A -85,B 0,C 180,E1 -6380.472,E2 -6380.472} C_VEL
LIN {X 0,Y 488.134,Z 652.752,A -85,B 0,C 180,E1 -6382.139,E2 -6382.139} C_VEL
LIN {X 0,Y 488.044,Z 656.367,A -85,B 0,C 180,E1 -6383.526,E2 -6383.526} C_VEL
LIN {X 0,Y 487.922,Z 659.405,A -85,B 0,C 180,E1 -6385.042,E2 -6385.042} C_VEL
LIN {X 0,Y 487.949,Z 661.856,A -85,B 0,C 180,E1 -6386.697,E2 -6386.697} C_VEL
LIN {X 0,Y 487.888,Z 663.255,A -85,B 0,C 180,E1 -6388.349,E2 -6388.349} C_VEL
LIN {X 0,Y 487.816,Z 663.798,A -85,B 0,C 180,E1 -6390,E2 -6390} C_VEL
LIN {X 0,Y 487.887,Z 663.307,A -85,B 0,C 180,E1 -6391.651,E2 -6391.651} C_VEL
LIN {X 0,Y 487.949,Z 661.959,A -85,B 0,C 180,E1 -6393.303,E2 -6393.303} C_VEL
LIN {X 0,Y 487.92,Z 659.561,A -85,B 0,C 180,E1 -6394.958,E2 -6394.958} C_VEL
LIN {X 0,Y 488.062,Z 656.247,A -85,B 0,C 180,E1 -6396.615,E2 -6396.615} C_VEL
LIN {X 0,Y 488.219,Z 650.557,A -85,B 0,C 180,E1 -6398.693,E2 -6398.693} C_VEL
LIN {X 0,Y 488.521,Z 643.071,A -85,B 0,C 180,E1 -6400.779,E2 -6400.779} C_VEL
LIN {X 0,Y 488.915,Z 634.586,A -85,B 0,C 180,E1 -6402.663,E2 -6402.663} C_VEL
LIN {X 0,Y 489.459,Z 625.428,A -85,B 0,C 180,E1 -6404.341,E2 -6404.341} C_VEL
LIN {X 0,Y 490.101,Z 614.988,A -85,B 0,C 180,E1 -6405.958,E2 -6405.958} C_VEL
LIN {X 0,Y 490.936,Z 603.242,A -85,B 0,C 180,E1 -6407.495,E2 -6407.495} C_VEL
LIN {X 0,Y 491.764,Z 590.938,A -85,B 0,C 180,E1 -6408.865,E2 -6408.865} C_VEL
LIN {X 0,Y 492.757,Z 577.523,A -85,B 0,C 180,E1 -6410.126,E2 -6410.126} C_VEL
LIN {X 0,Y 493.763,Z 562.753,A -85,B 0,C 180,E1 -6411.282,E2 -6411.282} C_VEL
LIN {X 0,Y 494.606,Z 548.826,A -85,B 0,C 180,E1 -6412.186,E2 -6412.186} C_VEL
LIN {X 0,Y 495.362,Z 534.421,A -85,B 0,C 180,E1 -6412.964,E2 -6412.964} C_VEL
LIN {X 0,Y 496.133,Z 518.508,A -85,B 0,C 180,E1 -6413.644,E2 -6413.644} C_VEL
LIN {X 0,Y 496.64,Z 502.893,A -85,B 0,C 180,E1 -6414.145,E2 -6414.145} C_VEL
LIN {X 0,Y 497.04,Z 486.201,A -85,B 0,C 180,E1 -6414.514,E2 -6414.514} C_VEL
LIN {X 0,Y 499.171,Z 303.186,A -85,B 0,C 180,E1 -6417.283,E2 -6417.283} C_VEL
LIN {X 0,Y 497.994,Z 298.149,A -85,B 0,C 180,E1 -6417.433,E2 -6417.433} C_VEL
LIN {X 0,Y 491.961,Z 284.956,A -85,B 0,C 180,E1 -6418.029,E2 -6418.029} C_VEL
LIN {X 0,Y 488.742,Z 273.911,A -85,B 0,C 180,E1 -6419.594,E2 -6419.594} C_VEL
LIN {X 0,Y 488.737,Z 273.912,A -85,B 0,C 180,E1 -6423.123,E2 -6423.123} C_VEL
LIN {X 0,Y 488.668,Z 273.915,A -85,B 0,C 180,E1 -6426.132,E2 -6426.132} C_VEL
LIN {X 0,Y 488.699,Z 273.924,A -85,B 0,C 180,E1 -6429.254,E2 -6429.254} C_VEL
LIN {X 0,Y 488.706,Z 273.92,A -85,B 0,C 180,E1 -6431.6,E2 -6431.6} C_VEL
LIN {X 0,Y 488.711,Z 273.921,A -85,B 0,C 180,E1 -6434.801,E2 -6434.801} C_VEL
LIN {X 0,Y 488.69,Z 273.924,A -85,B 0,C 180,E1 -6437.474,E2 -6437.474} C_VEL
LIN {X 0,Y 488.731,Z 273.917,A -85,B 0,C 180,E1 -6439.676,E2 -6439.676} C_VEL
LIN {X 0,Y 488.68,Z 273.921,A -85,B 0,C 180,E1 -6442.841,E2 -6442.841} C_VEL
LIN {X 0,Y 488.732,Z 273.914,A -85,B 0,C 180,E1 -6445.887,E2 -6445.887} C_VEL
LIN {X 0,Y 488.689,Z 273.92,A -85,B 0,C 180,E1 -6448.82,E2 -6448.82} C_VEL
LIN {X 0,Y 488.742,Z 273.908,A -85,B 0,C 180,E1 -6451.671,E2 -6451.671} C_VEL
LIN {X 0,Y 488.745,Z 273.913,A -85,B 0,C 180,E1 -6454.444,E2 -6454.444} C_VEL
LIN {X 0,Y 488.722,Z 273.913,A -85,B 0,C 180,E1 -6457.153,E2 -6457.153} C_VEL
LIN {X 0,Y 488.722,Z 273.916,A -85,B 0,C 180,E1 -6459.81,E2 -6459.81} C_VEL
LIN {X 0,Y 488.727,Z 273.915,A -85,B 0,C 180,E1 -6462.423,E2 -6462.423} C_VEL
LIN {X 0,Y 488.759,Z 273.907,A -85,B 0,C 180,E1 -6464.999,E2 -6464.999} C_VEL
LIN {X 0,Y 488.803,Z 273.906,A -85,B 0,C 180,E1 -6468.387,E2 -6468.387} C_VEL
LIN {X 0,Y 488.813,Z 273.902,A -85,B 0,C 180,E1 -6471.733,E2 -6471.733} C_VEL
LIN {X 0,Y 488.855,Z 273.9,A -85,B 0,C 180,E1 -6474.224,E2 -6474.224} C_VEL
LIN {X 0,Y 488.959,Z 273.881,A -85,B 0,C 180,E1 -6477.529,E2 -6477.529} C_VEL
LIN {X 0,Y 488.951,Z 273.893,A -85,B 0,C 180,E1 -6480.823,E2 -6480.823} C_VEL
LIN {X 0,Y 488.959,Z 273.887,A -85,B 0,C 180,E1 -6482.471,E2 -6482.471} C_VEL
LIN {X 0,Y 488.855,Z 273.898,A -85,B 0,C 180,E1 -6485.776,E2 -6485.776} C_VEL
LIN {X 0,Y 488.814,Z 273.905,A -85,B 0,C 180,E1 -6488.266,E2 -6488.266} C_VEL
LIN {X 0,Y 488.802,Z 273.903,A -85,B 0,C 180,E1 -6491.612,E2 -6491.612} C_VEL
LIN {X 0,Y 488.759,Z 273.916,A -85,B 0,C 180,E1 -6495,E2 -6495} C_VEL
LIN {X 0,Y 488.752,Z 273.914,A -85,B 0,C 180,E1 -6498.442,E2 -6498.442} C_VEL
LIN {X 0,Y 488.703,Z 273.923,A -85,B 0,C 180,E1 -6501.071,E2 -6501.071} C_VEL
LIN {X 0,Y 488.69,Z 273.921,A -85,B 0,C 180,E1 -6503.745,E2 -6503.745} C_VEL
LIN {X 0,Y 488.788,Z 273.914,A -85,B 0,C 180,E1 -6506.944,E2 -6506.944} C_VEL
LIN {X 0,Y 488.706,Z 273.922,A -85,B 0,C 180,E1 -6510.363,E2 -6510.363} C_VEL
LIN {X 0,Y 488.733,Z 273.919,A -85,B 0,C 180,E1 -6513.485,E2 -6513.485} C_VEL
LIN {X 0,Y 488.686,Z 273.924,A -85,B 0,C 180,E1 -6516.356,E2 -6516.356} C_VEL
LIN {X 0,Y 488.698,Z 273.925,A -85,B 0,C 180,E1 -6519.254,E2 -6519.254} C_VEL
LIN {X 0,Y 488.705,Z 273.922,A -85,B 0,C 180,E1 -6521.6,E2 -6521.6} C_VEL
LIN {X 0,Y 488.709,Z 273.927,A -85,B 0,C 180,E1 -6524.801,E2 -6524.801} C_VEL
LIN {X 0,Y 488.693,Z 273.923,A -85,B 0,C 180,E1 -6527.475,E2 -6527.475} C_VEL
LIN {X 0,Y 488.73,Z 273.917,A -85,B 0,C 180,E1 -6529.677,E2 -6529.677} C_VEL
LIN {X 0,Y 488.677,Z 273.926,A -85,B 0,C 180,E1 -6532.841,E2 -6532.841} C_VEL
LIN {X 0,Y 488.728,Z 273.909,A -85,B 0,C 180,E1 -6535.887,E2 -6535.887} C_VEL
LIN {X 0,Y 488.706,Z 273.968,A -85,B 0,C 180,E1 -6537.987,E2 -6537.987} C_VEL
LIN {X 0,Y 494.274,Z 292.105,A -85,B 0,C 180,E1 -6540.3,E2 -6540.3} C_VEL
LIN {X 0,Y 495.828,Z 297.759,A -85,B 0,C 180,E1 -6540.989,E2 -6540.989} C_VEL
LIN {X 0,Y 495.169,Z 310.301,A -85,B 0,C 180,E1 -6542.225,E2 -6542.225} C_VEL
LIN {X 0,Y 498.986,Z 332.236,A -85,B 0,C 180,E1 -6542.801,E2 -6542.801} C_VEL
LIN {X 0,Y 496.841,Z 516.201,A -85,B 0,C 180,E1 -6545.587,E2 -6545.587} C_VEL
LIN {X 0,Y 496.354,Z 531.54,A -85,B 0,C 180,E1 -6545.951,E2 -6545.951} C_VEL
LIN {X 0,Y 495.721,Z 547.953,A -85,B 0,C 180,E1 -6546.501,E2 -6546.501} C_VEL
LIN {X 0,Y 494.96,Z 563.472,A -85,B 0,C 180,E1 -6547.182,E2 -6547.182} C_VEL
LIN {X 0,Y 493.954,Z 580.066,A -85,B 0,C 180,E1 -6548.107,E2 -6548.107} C_VEL
LIN {X 0,Y 493.041,Z 594.756,A -85,B 0,C 180,E1 -6549.123,E2 -6549.123} C_VEL
LIN {X 0,Y 492.099,Z 608.755,A -85,B 0,C 180,E1 -6550.28,E2 -6550.28} C_VEL
LIN {X 0,Y 491.28,Z 620.751,A -85,B 0,C 180,E1 -6551.44,E2 -6551.44} C_VEL
LIN {X 0,Y 490.512,Z 631.998,A -85,B 0,C 180,E1 -6552.704,E2 -6552.704} C_VEL
LIN {X 0,Y 489.768,Z 643.218,A -85,B 0,C 180,E1 -6554.179,E2 -6554.179} C_VEL
LIN {X 0,Y 489.217,Z 652.853,A -85,B 0,C 180,E1 -6555.652,E2 -6555.652} C_VEL
LIN {X 0,Y 488.788,Z 662.224,A -85,B 0,C 180,E1 -6557.334,E2 -6557.334} C_VEL
LIN {X 0,Y 488.391,Z 670.905,A -85,B 0,C 180,E1 -6559.218,E2 -6559.218} C_VEL
LIN {X 0,Y 488.09,Z 678.594,A -85,B 0,C 180,E1 -6561.304,E2 -6561.304} C_VEL
LIN {X 0,Y 487.994,Z 684.447,A -85,B 0,C 180,E1 -6563.384,E2 -6563.384} C_VEL
LIN {X 0,Y 487.907,Z 687.868,A -85,B 0,C 180,E1 -6565.042,E2 -6565.042} C_VEL
LIN {X 0,Y 487.944,Z 690.357,A -85,B 0,C 180,E1 -6566.697,E2 -6566.697} C_VEL
LIN {X 0,Y 487.883,Z 691.759,A -85,B 0,C 180,E1 -6568.349,E2 -6568.349} C_VEL
LIN {X 0,Y 487.814,Z 692.286,A -85,B 0,C 180,E1 -6570,E2 -6570} C_VEL
LIN {X 0,Y 487.883,Z 691.759,A -85,B 0,C 180,E1 -6571.651,E2 -6571.651} C_VEL
LIN {X 0,Y 487.944,Z 690.356,A -85,B 0,C 180,E1 -6573.303,E2 -6573.303} C_VEL
LIN {X 0,Y 487.907,Z 687.867,A -85,B 0,C 180,E1 -6574.958,E2 -6574.958} C_VEL
LIN {X 0,Y 487.994,Z 684.45,A -85,B 0,C 180,E1 -6576.616,E2 -6576.616} C_VEL
LIN {X 0,Y 488.09,Z 678.597,A -85,B 0,C 180,E1 -6578.696,E2 -6578.696} C_VEL
LIN {X 0,Y 488.391,Z 670.905,A -85,B 0,C 180,E1 -6580.782,E2 -6580.782} C_VEL
LIN {X 0,Y 488.788,Z 662.224,A -85,B 0,C 180,E1 -6582.666,E2 -6582.666} C_VEL
LIN {X 0,Y 489.216,Z 652.855,A -85,B 0,C 180,E1 -6584.348,E2 -6584.348} C_VEL
LIN {X 0,Y 489.778,Z 643.219,A -85,B 0,C 180,E1 -6585.821,E2 -6585.821} C_VEL
LIN {X 0,Y 490.497,Z 631.996,A -85,B 0,C 180,E1 -6587.296,E2 -6587.296} C_VEL
LIN {X 0,Y 491.347,Z 619.768,A -85,B 0,C 180,E1 -6588.665,E2 -6588.665} C_VEL
LIN {X 0,Y 492.286,Z 606.403,A -85,B 0,C 180,E1 -6589.929,E2 -6589.929} C_VEL
LIN {X 0,Y 493.164,Z 593.322,A -85,B 0,C 180,E1 -6590.98,E2 -6590.98} C_VEL
LIN {X 0,Y 493.956,Z 580.08,A -85,B 0,C 180,E1 -6591.891,E2 -6591.891} C_VEL
LIN {X 0,Y 494.902,Z 564.461,A -85,B 0,C 180,E1 -6592.766,E2 -6592.766} C_VEL
LIN {X 0,Y 495.655,Z 549.253,A -85,B 0,C 180,E1 -6593.447,E2 -6593.447} C_VEL
LIN {X 0,Y 496.317,Z 532.452,A -85,B 0,C 180,E1 -6594.023,E2 -6594.023} C_VEL
LIN {X 0,Y 496.848,Z 516.181,A -85,B 0,C 180,E1 -6594.412,E2 -6594.412} C_VEL
LIN {X 0,Y 499.024,Z 332.128,A -85,B 0,C 180,E1 -6597.197,E2 -6597.197} C_VEL
LIN {X 0,Y 495.143,Z 309.866,A -85,B 0,C 180,E1 -6597.789,E2 -6597.789} C_VEL
LIN {X 0,Y 495.816,Z 297.736,A -85,B 0,C 180,E1 -6599.012,E2 -6599.012} C_VEL
LIN {X 0,Y 490.873,Z 280.807,A -85,B 0,C 180,E1 -6601.121,E2 -6601.121} C_VEL
LIN {X 0,Y 488.716,Z 273.923,A -85,B 0,C 180,E1 -6602.046,E2 -6602.046} C_VEL
LIN {X 0,Y 488.715,Z 273.923,A -85,B 0,C 180,E1 -6605.115,E2 -6605.115} C_VEL
LIN {X 0,Y 488.678,Z 273.924,A -85,B 0,C 180,E1 -6608.2,E2 -6608.2} C_VEL
LIN {X 0,Y 488.717,Z 273.924,A -85,B 0,C 180,E1 -6611.414,E2 -6611.414} C_VEL
LIN {X 0,Y 488.7,Z 273.918,A -85,B 0,C 180,E1 -6614.024,E2 -6614.024} C_VEL
LIN {X 0,Y 488.706,Z 273.923,A -85,B 0,C 180,E1 -6617.174,E2 -6617.174} C_VEL
LIN {X 0,Y 488.73,Z 273.915,A -85,B 0,C 180,E1 -6619.677,E2 -6619.677} C_VEL
LIN {X 0,Y 488.679,Z 273.922,A -85,B 0,C 180,E1 -6622.841,E2 -6622.841} C_VEL
LIN {X 0,Y 488.731,Z 273.915,A -85,B 0,C 180,E1 -6625.887,E2 -6625.887} C_VEL
LIN {X 0,Y 488.689,Z 273.923,A -85,B 0,C 180,E1 -6628.82,E2 -6628.82} C_VEL
LIN {X 0,Y 488.741,Z 273.915,A -85,B 0,C 180,E1 -6631.671,E2 -6631.671} C_VEL
LIN {X 0,Y 488.745,Z 273.914,A -85,B 0,C 180,E1 -6634.444,E2 -6634.444} C_VEL
LIN {X 0,Y 488.721,Z 273.924,A -85,B 0,C 180,E1 -6637.153,E2 -6637.153} C_VEL
LIN {X 0,Y 488.722,Z 273.905,A -85,B 0,C 180,E1 -6639.811,E2 -6639.811} C_VEL
LIN {X 0,Y 488.726,Z 273.915,A -85,B 0,C 180,E1 -6642.423,E2 -6642.423} C_VEL
LIN {X 0,Y 488.759,Z 273.911,A -85,B 0,C 180,E1 -6645,E2 -6645} C_VEL
LIN {X 0,Y 488.803,Z 273.903,A -85,B 0,C 180,E1 -6648.388,E2 -6648.388} C_VEL
LIN {X 0,Y 488.814,Z 273.9,A -85,B 0,C 180,E1 -6651.734,E2 -6651.734} C_VEL
LIN {X 0,Y 488.855,Z 273.888,A -85,B 0,C 180,E1 -6654.224,E2 -6654.224} C_VEL
LIN {X 0,Y 488.959,Z 273.888,A -85,B 0,C 180,E1 -6657.529,E2 -6657.529} C_VEL
LIN {X 0,Y 488.932,Z 273.881,A -85,B 0,C 180,E1 -6660.824,E2 -6660.824} C_VEL
LIN {X 0,Y 488.959,Z 273.881,A -85,B 0,C 180,E1 -6662.471,E2 -6662.471} C_VEL
LIN {X 0,Y 488.845,Z 273.899,A -85,B 0,C 180,E1 -6665.776,E2 -6665.776} C_VEL
LIN {X 0,Y 488.815,Z 273.89,A -85,B 0,C 180,E1 -6668.267,E2 -6668.267} C_VEL
LIN {X 0,Y 488.803,Z 273.907,A -85,B 0,C 180,E1 -6671.613,E2 -6671.613} C_VEL
LIN {X 0,Y 488.76,Z 273.904,A -85,B 0,C 180,E1 -6675.001,E2 -6675.001} C_VEL
LIN {X 0,Y 488.753,Z 273.914,A -85,B 0,C 180,E1 -6678.442,E2 -6678.442} C_VEL
LIN {X 0,Y 488.705,Z 273.912,A -85,B 0,C 180,E1 -6681.071,E2 -6681.071} C_VEL
LIN {X 0,Y 488.691,Z 273.919,A -85,B 0,C 180,E1 -6683.746,E2 -6683.746} C_VEL
LIN {X 0,Y 488.79,Z 273.904,A -85,B 0,C 180,E1 -6686.944,E2 -6686.944} C_VEL
LIN {X 0,Y 488.708,Z 273.919,A -85,B 0,C 180,E1 -6690.363,E2 -6690.363} C_VEL
LIN {X 0,Y 488.734,Z 273.915,A -85,B 0,C 180,E1 -6693.485,E2 -6693.485} C_VEL
LIN {X 0,Y 488.688,Z 273.922,A -85,B 0,C 180,E1 -6696.356,E2 -6696.356} C_VEL
LIN {X 0,Y 488.7,Z 273.921,A -85,B 0,C 180,E1 -6699.254,E2 -6699.254} C_VEL
LIN {X 0,Y 488.706,Z 273.913,A -85,B 0,C 180,E1 -6701.6,E2 -6701.6} C_VEL
LIN {X 0,Y 488.711,Z 273.922,A -85,B 0,C 180,E1 -6704.802,E2 -6704.802} C_VEL
LIN {X 0,Y 488.691,Z 273.922,A -85,B 0,C 180,E1 -6707.475,E2 -6707.475} C_VEL
LIN {X 0,Y 488.732,Z 273.916,A -85,B 0,C 180,E1 -6709.677,E2 -6709.677} C_VEL
LIN {X 0,Y 488.678,Z 273.912,A -85,B 0,C 180,E1 -6712.841,E2 -6712.841} C_VEL
LIN {X 0,Y 488.73,Z 273.916,A -85,B 0,C 180,E1 -6715.887,E2 -6715.887} C_VEL
LIN {X 0,Y 488.692,Z 273.926,A -85,B 0,C 180,E1 -6718.821,E2 -6718.821} C_VEL
LIN {X 0,Y 488.732,Z 273.965,A -85,B 0,C 180,E1 -6720.524,E2 -6720.524} C_VEL
LIN {X 0,Y 492.083,Z 285.191,A -85,B 0,C 180,E1 -6722.088,E2 -6722.088} C_VEL
LIN {X 0,Y 494.095,Z 289.637,A -85,B 0,C 180,E1 -6722.284,E2 -6722.284} C_VEL
LIN {X 0,Y 495.06,Z 293.307,A -85,B 0,C 180,E1 -6722.403,E2 -6722.403} C_VEL
LIN {X 0,Y 495.39,Z 299.147,A -85,B 0,C 180,E1 -6722.516,E2 -6722.516} C_VEL
LIN {X 0,Y 494.831,Z 305.083,A -85,B 0,C 180,E1 -6722.578,E2 -6722.578} C_VEL
LIN {X 0,Y 492.953,Z 317.263,A -85,B 0,C 180,E1 -6722.66,E2 -6722.66} C_VEL
LIN {X 0,Y 492.669,Z 321.337,A -85,B 0,C 180,E1 -6722.708,E2 -6722.708} C_VEL
LIN {X 0,Y 490.627,Z 487.553,A -85,B 0,C 180,E1 -6725.257,E2 -6725.257} C_VEL
LIN {X 0,Y 490.196,Z 502.883,A -85,B 0,C 180,E1 -6725.601,E2 -6725.601} C_VEL
LIN {X 0,Y 489.601,Z 519.253,A -85,B 0,C 180,E1 -6726.133,E2 -6726.133} C_VEL
LIN {X 0,Y 488.818,Z 534.693,A -85,B 0,C 180,E1 -6726.806,E2 -6726.806} C_VEL
LIN {X 0,Y 488.003,Z 549.146,A -85,B 0,C 180,E1 -6727.596,E2 -6727.596} C_VEL
LIN {X 0,Y 487.072,Z 563.214,A -85,B 0,C 180,E1 -6728.523,E2 -6728.523} C_VEL
LIN {X 0,Y 486.094,Z 576.693,A -85,B 0,C 180,E1 -6729.586,E2 -6729.586} C_VEL
LIN {X 0,Y 485.089,Z 590.266,A -85,B 0,C 180,E1 -6730.865,E2 -6730.865} C_VEL
LIN {X 0,Y 484.132,Z 602.714,A -85,B 0,C 180,E1 -6732.251,E2 -6732.251} C_VEL
LIN {X 0,Y 483.254,Z 614.864,A -85,B 0,C 180,E1 -6733.852,E2 -6733.852} C_VEL
LIN {X 0,Y 482.557,Z 625.124,A -85,B 0,C 180,E1 -6735.45,E2 -6735.45} C_VEL
LIN {X 0,Y 481.971,Z 634.363,A -85,B 0,C 180,E1 -6737.152,E2 -6737.152} C_VEL
LIN {X 0,Y 481.525,Z 642.905,A -85,B 0,C 180,E1 -6739.063,E2 -6739.063} C_VEL
LIN {X 0,Y 481.153,Z 650.483,A -85,B 0,C 180,E1 -6741.178,E2 -6741.178} C_VEL
LIN {X 0,Y 480.994,Z 656.237,A -85,B 0,C 180,E1 -6743.287,E2 -6743.287} C_VEL
LIN {X 0,Y 480.852,Z 659.613,A -85,B 0,C 180,E1 -6744.969,E2 -6744.969} C_VEL
LIN {X 0,Y 480.874,Z 662.063,A -85,B 0,C 180,E1 -6746.649,E2 -6746.649} C_VEL
LIN {X 0,Y 480.819,Z 663.462,A -85,B 0,C 180,E1 -6748.325,E2 -6748.325} C_VEL
LIN {X 0,Y 480.74,Z 664.004,A -85,B 0,C 180,E1 -6750,E2 -6750} C_VEL
LIN {X 0,Y 480.818,Z 663.513,A -85,B 0,C 180,E1 -6751.675,E2 -6751.675} C_VEL
LIN {X 0,Y 480.874,Z 662.166,A -85,B 0,C 180,E1 -6753.351,E2 -6753.351} C_VEL
LIN {X 0,Y 480.851,Z 659.767,A -85,B 0,C 180,E1 -6755.031,E2 -6755.031} C_VEL
LIN {X 0,Y 480.994,Z 656.453,A -85,B 0,C 180,E1 -6756.713,E2 -6756.713} C_VEL
LIN {X 0,Y 481.145,Z 650.764,A -85,B 0,C 180,E1 -6758.822,E2 -6758.822} C_VEL
LIN {X 0,Y 481.483,Z 643.277,A -85,B 0,C 180,E1 -6760.938,E2 -6760.938} C_VEL
LIN {X 0,Y 481.918,Z 634.792,A -85,B 0,C 180,E1 -6762.85,E2 -6762.85} C_VEL
LIN {X 0,Y 482.532,Z 625.633,A -85,B 0,C 180,E1 -6764.551,E2 -6764.551} C_VEL
LIN {X 0,Y 483.141,Z 616.209,A -85,B 0,C 180,E1 -6766.044,E2 -6766.044} C_VEL
LIN {X 0,Y 483.987,Z 605.215,A -85,B 0,C 180,E1 -6767.536,E2 -6767.536} C_VEL
LIN {X 0,Y 484.932,Z 592.199,A -85,B 0,C 180,E1 -6769.031,E2 -6769.031} C_VEL
LIN {X 0,Y 485.963,Z 578.899,A -85,B 0,C 180,E1 -6770.309,E2 -6770.309} C_VEL
LIN {X 0,Y 486.894,Z 565.794,A -85,B 0,C 180,E1 -6771.375,E2 -6771.375} C_VEL
LIN {X 0,Y 487.895,Z 550.978,A -85,B 0,C 180,E1 -6772.384,E2 -6772.384} C_VEL
LIN {X 0,Y 488.696,Z 536.613,A -85,B 0,C 180,E1 -6773.195,E2 -6773.195} C_VEL
LIN {X 0,Y 489.512,Z 521.353,A -85,B 0,C 180,E1 -6773.872,E2 -6773.872} C_VEL
LIN {X 0,Y 490.087,Z 505.826,A -85,B 0,C 180,E1 -6774.405,E2 -6774.405} C_VEL
LIN {X 0,Y 490.561,Z 490.89,A -85,B 0,C 180,E1 -6774.774,E2 -6774.774} C_VEL
LIN {X 0,Y 492.872,Z 304.48,A -85,B 0,C 180,E1 -6777.643,E2 -6777.643} C_VEL
LIN {X 0,Y 491.877,Z 300.604,A -85,B 0,C 180,E1 -6777.767,E2 -6777.767} C_VEL
LIN {X 0,Y 484.801,Z 285.281,A -85,B 0,C 180,E1 -6778.468,E2 -6778.468} C_VEL
LIN {X 0,Y 481.673,Z 274.792,A -85,B 0,C 180,E1 -6779.982,E2 -6779.982} C_VEL
LIN {X 0,Y 481.671,Z 274.791,A -85,B 0,C 180,E1 -6782.674,E2 -6782.674} C_VEL
LIN {X 0,Y 481.659,Z 274.799,A -85,B 0,C 180,E1 -6785.204,E2 -6785.204} C_VEL
LIN {X 0,Y 481.669,Z 274.8,A -85,B 0,C 180,E1 -6788.859,E2 -6788.859} C_VEL
LIN {X 0,Y 481.651,Z 274.796,A -85,B 0,C 180,E1 -6791.913,E2 -6791.913} C_VEL
LIN {X 0,Y 481.658,Z 274.798,A -85,B 0,C 180,E1 -6794.457,E2 -6794.457} C_VEL
LIN {X 0,Y 481.646,Z 274.798,A -85,B 0,C 180,E1 -6797.839,E2 -6797.839} C_VEL
LIN {X 0,Y 481.659,Z 274.797,A -85,B 0,C 180,E1 -6800.654,E2 -6800.654} C_VEL
LIN {X 0,Y 481.628,Z 274.8,A -85,B 0,C 180,E1 -6803.375,E2 -6803.375} C_VEL
LIN {X 0,Y 481.708,Z 274.789,A -85,B 0,C 180,E1 -6806.33,E2 -6806.33} C_VEL
LIN {X 0,Y 481.648,Z 274.803,A -85,B 0,C 180,E1 -6809.417,E2 -6809.417} C_VEL
LIN {X 0,Y 481.697,Z 274.783,A -85,B 0,C 180,E1 -6812.168,E2 -6812.168} C_VEL
LIN {X 0,Y 481.716,Z 274.794,A -85,B 0,C 180,E1 -6814.97,E2 -6814.97} C_VEL
LIN {X 0,Y 481.647,Z 274.788,A -85,B 0,C 180,E1 -6817.705,E2 -6817.705} C_VEL
LIN {X 0,Y 481.702,Z 274.791,A -85,B 0,C 180,E1 -6820.393,E2 -6820.393} C_VEL
LIN {X 0,Y 481.686,Z 274.789,A -85,B 0,C 180,E1 -6823.034,E2 -6823.034} C_VEL
LIN {X 0,Y 481.687,Z 274.793,A -85,B 0,C 180,E1 -6825.639,E2 -6825.639} C_VEL
LIN {X 0,Y 481.748,Z 274.784,A -85,B 0,C 180,E1 -6828.215,E2 -6828.215} C_VEL
LIN {X 0,Y 481.759,Z 274.781,A -85,B 0,C 180,E1 -6831.612,E2 -6831.612} C_VEL
LIN {X 0,Y 481.816,Z 274.777,A -85,B 0,C 180,E1 -6834.139,E2 -6834.139} C_VEL
LIN {X 0,Y 481.926,Z 274.756,A -85,B 0,C 180,E1 -6837.492,E2 -6837.492} C_VEL
LIN {X 0,Y 481.902,Z 274.772,A -85,B 0,C 180,E1 -6840.835,E2 -6840.835} C_VEL
LIN {X 0,Y 481.925,Z 274.763,A -85,B 0,C 180,E1 -6842.507,E2 -6842.507} C_VEL
LIN {X 0,Y 481.816,Z 274.774,A -85,B 0,C 180,E1 -6845.86,E2 -6845.86} C_VEL
LIN {X 0,Y 481.76,Z 274.785,A -85,B 0,C 180,E1 -6848.388,E2 -6848.388} C_VEL
LIN {X 0,Y 481.748,Z 274.781,A -85,B 0,C 180,E1 -6851.785,E2 -6851.785} C_VEL
LIN {X 0,Y 481.739,Z 274.79,A -85,B 0,C 180,E1 -6855.224,E2 -6855.224} C_VEL
LIN {X 0,Y 481.709,Z 274.794,A -85,B 0,C 180,E1 -6858.722,E2 -6858.722} C_VEL
LIN {X 0,Y 481.642,Z 274.8,A -85,B 0,C 180,E1 -6861.395,E2 -6861.395} C_VEL
LIN {X 0,Y 481.674,Z 274.795,A -85,B 0,C 180,E1 -6864.113,E2 -6864.113} C_VEL
LIN {X 0,Y 481.743,Z 274.791,A -85,B 0,C 180,E1 -6867.139,E2 -6867.139} C_VEL
LIN {X 0,Y 481.675,Z 274.795,A -85,B 0,C 180,E1 -6869.741,E2 -6869.741} C_VEL
LIN {X 0,Y 481.669,Z 274.802,A -85,B 0,C 180,E1 -6872.674,E2 -6872.674} C_VEL
LIN {X 0,Y 481.64,Z 274.799,A -85,B 0,C 180,E1 -6875.709,E2 -6875.709} C_VEL
LIN {X 0,Y 481.668,Z 274.804,A -85,B 0,C 180,E1 -6878.859,E2 -6878.859} C_VEL
LIN {X 0,Y 481.65,Z 274.801,A -85,B 0,C 180,E1 -6881.913,E2 -6881.913} C_VEL
LIN {X 0,Y 481.657,Z 274.804,A -85,B 0,C 180,E1 -6884.457,E2 -6884.457} C_VEL
LIN {X 0,Y 481.651,Z 274.8,A -85,B 0,C 180,E1 -6887.84,E2 -6887.84} C_VEL
LIN {X 0,Y 481.678,Z 274.801,A -85,B 0,C 180,E1 -6890.651,E2 -6890.651} C_VEL
LIN {X 0,Y 481.625,Z 274.805,A -85,B 0,C 180,E1 -6893.376,E2 -6893.376} C_VEL
LIN {X 0,Y 481.707,Z 274.788,A -85,B 0,C 180,E1 -6896.33,E2 -6896.33} C_VEL
LIN {X 0,Y 481.685,Z 274.898,A -85,B 0,C 180,E1 -6897.59,E2 -6897.59} C_VEL
LIN {X 0,Y 487.226,Z 292.913,A -85,B 0,C 180,E1 -6899.936,E2 -6899.936} C_VEL
LIN {X 0,Y 489.097,Z 299.462,A -85,B 0,C 180,E1 -6900.754,E2 -6900.754} C_VEL
LIN {X 0,Y 488.604,Z 309.727,A -85,B 0,C 180,E1 -6901.812,E2 -6901.812} C_VEL
LIN {X 0,Y 492.591,Z 332.087,A -85,B 0,C 180,E1 -6902.419,E2 -6902.419} C_VEL
LIN {X 0,Y 491.111,Z 458.261,A -85,B 0,C 180,E1 -6904.349,E2 -6904.349} C_VEL
LIN {X 0,Y 490.33,Z 517.642,A -85,B 0,C 180,E1 -6905.273,E2 -6905.273} C_VEL
LIN {X 0,Y 489.821,Z 533.174,A -85,B 0,C 180,E1 -6905.666,E2 -6905.666} C_VEL
LIN {X 0,Y 489.113,Z 549.053,A -85,B 0,C 180,E1 -6906.22,E2 -6906.22} C_VEL
LIN {X 0,Y 488.32,Z 564.266,A -85,B 0,C 180,E1 -6906.91,E2 -6906.91} C_VEL
LIN {X 0,Y 487.317,Z 580.071,A -85,B 0,C 180,E1 -6907.807,E2 -6907.807} C_VEL
LIN {X 0,Y 486.33,Z 594.548,A -85,B 0,C 180,E1 -6908.822,E2 -6908.822} C_VEL
LIN {X 0,Y 485.429,Z 607.382,A -85,B 0,C 180,E1 -6909.888,E2 -6909.888} C_VEL
LIN {X 0,Y 484.42,Z 620.54,A -85,B 0,C 180,E1 -6911.168,E2 -6911.168} C_VEL
LIN {X 0,Y 483.618,Z 631.787,A -85,B 0,C 180,E1 -6912.45,E2 -6912.45} C_VEL
LIN {X 0,Y 482.854,Z 643.008,A -85,B 0,C 180,E1 -6913.946,E2 -6913.946} C_VEL
LIN {X 0,Y 482.229,Z 652.643,A -85,B 0,C 180,E1 -6915.44,E2 -6915.44} C_VEL
LIN {X 0,Y 481.75,Z 662.013,A -85,B 0,C 180,E1 -6917.146,E2 -6917.146} C_VEL
LIN {X 0,Y 481.428,Z 668.87,A -85,B 0,C 180,E1 -6918.634,E2 -6918.634} C_VEL
LIN {X 0,Y 481.075,Z 675.513,A -85,B 0,C 180,E1 -6920.328,E2 -6920.328} C_VEL
LIN {X 0,Y 480.985,Z 680.907,A -85,B 0,C 180,E1 -6922.021,E2 -6922.021} C_VEL
LIN {X 0,Y 480.911,Z 684.906,A -85,B 0,C 180,E1 -6923.587,E2 -6923.587} C_VEL
LIN {X 0,Y 480.832,Z 687.66,A -85,B 0,C 180,E1 -6924.969,E2 -6924.969} C_VEL
LIN {X 0,Y 480.867,Z 690.15,A -85,B 0,C 180,E1 -6926.649,E2 -6926.649} C_VEL
LIN {X 0,Y 480.784,Z 691.552,A -85,B 0,C 180,E1 -6928.325,E2 -6928.325} C_VEL
LIN {X 0,Y 480.738,Z 692.08,A -85,B 0,C 180,E1 -6930,E2 -6930} C_VEL
LIN {X 0,Y 480.784,Z 691.551,A -85,B 0,C 180,E1 -6931.675,E2 -6931.675} C_VEL
LIN {X 0,Y 480.867,Z 690.149,A -85,B 0,C 180,E1 -6933.351,E2 -6933.351} C_VEL
LIN {X 0,Y 480.832,Z 687.66,A -85,B 0,C 180,E1 -6935.031,E2 -6935.031} C_VEL
LIN {X 0,Y 480.904,Z 684.241,A -85,B 0,C 180,E1 -6936.714,E2 -6936.714} C_VEL
LIN {X 0,Y 481.03,Z 678.389,A -85,B 0,C 180,E1 -6938.824,E2 -6938.824} C_VEL
LIN {X 0,Y 481.325,Z 670.695,A -85,B 0,C 180,E1 -6940.942,E2 -6940.942} C_VEL
LIN {X 0,Y 481.724,Z 663.033,A -85,B 0,C 180,E1 -6942.641,E2 -6942.641} C_VEL
LIN {X 0,Y 482.149,Z 653.886,A -85,B 0,C 180,E1 -6944.347,E2 -6944.347} C_VEL
LIN {X 0,Y 482.77,Z 644.506,A -85,B 0,C 180,E1 -6945.84,E2 -6945.84} C_VEL
LIN {X 0,Y 483.499,Z 633.521,A -85,B 0,C 180,E1 -6947.336,E2 -6947.336} C_VEL
LIN {X 0,Y 484.319,Z 622.502,A -85,B 0,C 180,E1 -6948.617,E2 -6948.617} C_VEL
LIN {X 0,Y 485.3,Z 608.539,A -85,B 0,C 180,E1 -6950.009,E2 -6950.009} C_VEL
LIN {X 0,Y 486.362,Z 594.544,A -85,B 0,C 180,E1 -6951.177,E2 -6951.177} C_VEL
LIN {X 0,Y 487.31,Z 580.099,A -85,B 0,C 180,E1 -6952.19,E2 -6952.19} C_VEL
LIN {X 0,Y 488.314,Z 564.249,A -85,B 0,C 180,E1 -6953.091,E2 -6953.091} C_VEL
LIN {X 0,Y 489.133,Z 549.041,A -85,B 0,C 180,E1 -6953.779,E2 -6953.779} C_VEL
LIN {X 0,Y 489.817,Z 532.238,A -85,B 0,C 180,E1 -6954.363,E2 -6954.363} C_VEL
LIN {X 0,Y 490.39,Z 516.196,A -85,B 0,C 180,E1 -6954.751,E2 -6954.751} C_VEL
LIN {X 0,Y 492.674,Z 332.185,A -85,B 0,C 180,E1 -6957.573,E2 -6957.573} C_VEL
LIN {X 0,Y 488.573,Z 309.709,A -85,B 0,C 180,E1 -6958.19,E2 -6958.19} C_VEL
LIN {X 0,Y 489.095,Z 299.442,A -85,B 0,C 180,E1 -6959.246,E2 -6959.246} C_VEL
LIN {X 0,Y 483.767,Z 281.472,A -85,B 0,C 180,E1 -6961.533,E2 -6961.533} C_VEL
LIN {X 0,Y 481.67,Z 274.8,A -85,B 0,C 180,E1 -6962.429,E2 -6962.429} C_VEL
LIN {X 0,Y 481.66,Z 274.802,A -85,B 0,C 180,E1 -6965.204,E2 -6965.204} C_VEL
LIN {X 0,Y 481.669,Z 274.8,A -85,B 0,C 180,E1 -6968.859,E2 -6968.859} C_VEL
LIN {X 0,Y 481.66,Z 274.798,A -85,B 0,C 180,E1 -6971.914,E2 -6971.914} C_VEL
LIN {X 0,Y 481.658,Z 274.795,A -85,B 0,C 180,E1 -6974.457,E2 -6974.457} C_VEL
LIN {X 0,Y 481.645,Z 274.796,A -85,B 0,C 180,E1 -6977.839,E2 -6977.839} C_VEL
LIN {X 0,Y 481.658,Z 274.794,A -85,B 0,C 180,E1 -6980.654,E2 -6980.654} C_VEL
LIN {X 0,Y 481.628,Z 274.805,A -85,B 0,C 180,E1 -6983.376,E2 -6983.376} C_VEL
LIN {X 0,Y 481.707,Z 274.789,A -85,B 0,C 180,E1 -6986.33,E2 -6986.33} C_VEL
LIN {X 0,Y 481.648,Z 274.8,A -85,B 0,C 180,E1 -6989.417,E2 -6989.417} C_VEL
LIN {X 0,Y 481.697,Z 274.79,A -85,B 0,C 180,E1 -6992.168,E2 -6992.168} C_VEL
LIN {X 0,Y 481.716,Z 274.795,A -85,B 0,C 180,E1 -6994.97,E2 -6994.97} C_VEL
LIN {X 0,Y 481.647,Z 274.798,A -85,B 0,C 180,E1 -6997.705,E2 -6997.705} C_VEL
LIN {X 0,Y 481.702,Z 274.778,A -85,B 0,C 180,E1 -7000.393,E2 -7000.393} C_VEL
LIN {X 0,Y 481.685,Z 274.799,A -85,B 0,C 180,E1 -7003.034,E2 -7003.034} C_VEL
LIN {X 0,Y 481.686,Z 274.783,A -85,B 0,C 180,E1 -7005.639,E2 -7005.639} C_VEL
LIN {X 0,Y 481.748,Z 274.781,A -85,B 0,C 180,E1 -7008.215,E2 -7008.215} C_VEL
LIN {X 0,Y 481.76,Z 274.78,A -85,B 0,C 180,E1 -7011.612,E2 -7011.612} C_VEL
LIN {X 0,Y 481.816,Z 274.764,A -85,B 0,C 180,E1 -7014.14,E2 -7014.14} C_VEL
LIN {X 0,Y 481.926,Z 274.765,A -85,B 0,C 180,E1 -7017.493,E2 -7017.493} C_VEL
LIN {X 0,Y 481.884,Z 274.758,A -85,B 0,C 180,E1 -7020.836,E2 -7020.836} C_VEL
LIN {X 0,Y 481.926,Z 274.757,A -85,B 0,C 180,E1 -7022.508,E2 -7022.508} C_VEL
LIN {X 0,Y 481.806,Z 274.775,A -85,B 0,C 180,E1 -7025.861,E2 -7025.861} C_VEL
LIN {X 0,Y 481.76,Z 274.769,A -85,B 0,C 180,E1 -7028.388,E2 -7028.388} C_VEL
LIN {X 0,Y 481.749,Z 274.785,A -85,B 0,C 180,E1 -7031.785,E2 -7031.785} C_VEL
LIN {X 0,Y 481.74,Z 274.777,A -85,B 0,C 180,E1 -7035.224,E2 -7035.224} C_VEL
LIN {X 0,Y 481.71,Z 274.795,A -85,B 0,C 180,E1 -7038.722,E2 -7038.722} C_VEL
LIN {X 0,Y 481.643,Z 274.787,A -85,B 0,C 180,E1 -7041.395,E2 -7041.395} C_VEL
LIN {X 0,Y 481.675,Z 274.793,A -85,B 0,C 180,E1 -7044.113,E2 -7044.113} C_VEL
LIN {X 0,Y 481.745,Z 274.778,A -85,B 0,C 180,E1 -7047.139,E2 -7047.139} C_VEL
LIN {X 0,Y 481.677,Z 274.794,A -85,B 0,C 180,E1 -7049.741,E2 -7049.741} C_VEL
LIN {X 0,Y 481.67,Z 274.798,A -85,B 0,C 180,E1 -7052.674,E2 -7052.674} C_VEL
LIN {X 0,Y 481.641,Z 274.798,A -85,B 0,C 180,E1 -7055.709,E2 -7055.709} C_VEL
LIN {X 0,Y 481.669,Z 274.792,A -85,B 0,C 180,E1 -7058.859,E2 -7058.859} C_VEL
LIN {X 0,Y 481.651,Z 274.791,A -85,B 0,C 180,E1 -7061.913,E2 -7061.913} C_VEL
LIN {X 0,Y 481.659,Z 274.8,A -85,B 0,C 180,E1 -7064.458,E2 -7064.458} C_VEL
LIN {X 0,Y 481.647,Z 274.799,A -85,B 0,C 180,E1 -7067.84,E2 -7067.84} C_VEL
LIN {X 0,Y 481.68,Z 274.801,A -85,B 0,C 180,E1 -7070.651,E2 -7070.651} C_VEL
LIN {X 0,Y 481.626,Z 274.792,A -85,B 0,C 180,E1 -7073.376,E2 -7073.376} C_VEL
LIN {X 0,Y 481.709,Z 274.785,A -85,B 0,C 180,E1 -7076.33,E2 -7076.33} C_VEL
LIN {X 0,Y 481.692,Z 274.797,A -85,B 0,C 180,E1 -7079.777,E2 -7079.777} C_VEL
LIN {X 0,Y 481.7,Z 274.909,A -85,B 0,C 180,E1 -7080.14,E2 -7080.14} C_VEL
LIN {X 0,Y 484.919,Z 285.641,A -85,B 0,C 180,E1 -7081.642,E2 -7081.642} C_VEL
LIN {X 0,Y 492.481,Z 302.266,A -85,B 0,C 180,E1 -7082.389,E2 -7082.389} C_VEL
LIN {X 0,Y 492.897,Z 306.271,A -85,B 0,C 180,E1 -7082.479,E2 -7082.479} C_VEL
LIN {X 0,Y 492.669,Z 321.337,A -85,B 0,C 180,E1 -7082.708,E2 -7082.708} C_VEL
LIN {X 0,Y 491.951,Z 327.195,A -85,B 0,C 180,E1 -7082.759,E2 -7082.759} C_VEL
LIN {X 0,Y 486.59,Z 346.302,A -85,B 0,C 180,E1 -7082.742,E2 -7082.742} C_VEL
LIN {X 0,Y 485.977,Z 352.152,A -85,B 0,C 180,E1 -7082.8,E2 -7082.8} C_VEL
LIN {X 0,Y 484.199,Z 487.785,A -85,B 0,C 180,E1 -7084.906,E2 -7084.906} C_VEL
LIN {X 0,Y 483.761,Z 503.105,A -85,B 0,C 180,E1 -7085.255,E2 -7085.255} C_VEL
LIN {X 0,Y 483.122,Z 519.471,A -85,B 0,C 180,E1 -7085.793,E2 -7085.793} C_VEL
LIN {X 0,Y 482.306,Z 534.909,A -85,B 0,C 180,E1 -7086.474,E2 -7086.474} C_VEL
LIN {X 0,Y 481.412,Z 549.638,A -85,B 0,C 180,E1 -7087.29,E2 -7087.29} C_VEL
LIN {X 0,Y 480.455,Z 563.428,A -85,B 0,C 180,E1 -7088.212,E2 -7088.212} C_VEL
LIN {X 0,Y 479.317,Z 578.157,A -85,B 0,C 180,E1 -7089.397,E2 -7089.397} C_VEL
LIN {X 0,Y 478.263,Z 591.541,A -85,B 0,C 180,E1 -7090.693,E2 -7090.693} C_VEL
LIN {X 0,Y 477.301,Z 602.928,A -85,B 0,C 180,E1 -7091.988,E2 -7091.988} C_VEL
LIN {X 0,Y 476.438,Z 614.317,A -85,B 0,C 180,E1 -7093.501,E2 -7093.501} C_VEL
LIN {X 0,Y 475.699,Z 624.103,A -85,B 0,C 180,E1 -7095.016,E2 -7095.016} C_VEL
LIN {X 0,Y 475.043,Z 633.477,A -85,B 0,C 180,E1 -7096.743,E2 -7096.743} C_VEL
LIN {X 0,Y 474.582,Z 641.327,A -85,B 0,C 180,E1 -7098.468,E2 -7098.468} C_VEL
LIN {X 0,Y 474.177,Z 647.879,A -85,B 0,C 180,E1 -7100.186,E2 -7100.186} C_VEL
LIN {X 0,Y 474.012,Z 653.172,A -85,B 0,C 180,E1 -7101.903,E2 -7101.903} C_VEL
LIN {X 0,Y 473.88,Z 657.225,A -85,B 0,C 180,E1 -7103.545,E2 -7103.545} C_VEL
LIN {X 0,Y 473.727,Z 661.166,A -85,B 0,C 180,E1 -7105.746,E2 -7105.746} C_VEL
LIN {X 0,Y 473.754,Z 663.077,A -85,B 0,C 180,E1 -7107.449,E2 -7107.449} C_VEL
LIN {X 0,Y 473.685,Z 664.053,A -85,B 0,C 180,E1 -7109.15,E2 -7109.15} C_VEL
LIN {X 0,Y 473.684,Z 664.07,A -85,B 0,C 180,E1 -7110.85,E2 -7110.85} C_VEL
LIN {X 0,Y 473.754,Z 663.162,A -85,B 0,C 180,E1 -7112.551,E2 -7112.551} C_VEL
LIN {X 0,Y 473.725,Z 661.285,A -85,B 0,C 180,E1 -7114.254,E2 -7114.254} C_VEL
LIN {X 0,Y 473.876,Z 658.435,A -85,B 0,C 180,E1 -7115.959,E2 -7115.959} C_VEL
LIN {X 0,Y 473.966,Z 654.558,A -85,B 0,C 180,E1 -7117.669,E2 -7117.669} C_VEL
LIN {X 0,Y 474.128,Z 649.578,A -85,B 0,C 180,E1 -7119.384,E2 -7119.384} C_VEL
LIN {X 0,Y 474.46,Z 643.484,A -85,B 0,C 180,E1 -7121.102,E2 -7121.102} C_VEL
LIN {X 0,Y 474.94,Z 634.998,A -85,B 0,C 180,E1 -7123.042,E2 -7123.042} C_VEL
LIN {X 0,Y 475.601,Z 625.839,A -85,B 0,C 180,E1 -7124.768,E2 -7124.768} C_VEL
LIN {X 0,Y 476.276,Z 616.414,A -85,B 0,C 180,E1 -7126.282,E2 -7126.282} C_VEL
LIN {X 0,Y 477.156,Z 605.42,A -85,B 0,C 180,E1 -7127.796,E2 -7127.796} C_VEL
LIN {X 0,Y 478.185,Z 592.402,A -85,B 0,C 180,E1 -7129.31,E2 -7129.31} C_VEL
LIN {X 0,Y 479.281,Z 579.102,A -85,B 0,C 180,E1 -7130.605,E2 -7130.605} C_VEL
LIN {X 0,Y 480.277,Z 565.995,A -85,B 0,C 180,E1 -7131.684,E2 -7131.684} C_VEL
LIN {X 0,Y 481.297,Z 551.517,A -85,B 0,C 180,E1 -7132.686,E2 -7132.686} C_VEL
LIN {X 0,Y 482.172,Z 537.041,A -85,B 0,C 180,E1 -7133.516,E2 -7133.516} C_VEL
LIN {X 0,Y 483.016,Z 521.55,A -85,B 0,C 180,E1 -7134.213,E2 -7134.213} C_VEL
LIN {X 0,Y 483.663,Z 505.104,A -85,B 0,C 180,E1 -7134.779,E2 -7134.779} C_VEL
LIN {X 0,Y 484.166,Z 488.223,A -85,B 0,C 180,E1 -7135.178,E2 -7135.178} C_VEL
LIN {X 0,Y 486.6,Z 305.646,A -85,B 0,C 180,E1 -7138.014,E2 -7138.014} C_VEL
LIN {X 0,Y 485.642,Z 302.704,A -85,B 0,C 180,E1 -7138.123,E2 -7138.123} C_VEL
LIN {X 0,Y 477.522,Z 285.288,A -85,B 0,C 180,E1 -7138.97,E2 -7138.97} C_VEL
LIN {X 0,Y 474.623,Z 275.674,A -85,B 0,C 180,E1 -7140.399,E2 -7140.399} C_VEL
LIN {X 0,Y 474.642,Z 275.667,A -85,B 0,C 180,E1 -7143.22,E2 -7143.22} C_VEL
LIN {X 0,Y 474.583,Z 275.667,A -85,B 0,C 180,E1 -7146.324,E2 -7146.324} C_VEL
LIN {X 0,Y 474.616,Z 275.675,A -85,B 0,C 180,E1 -7149.646,E2 -7149.646} C_VEL
LIN {X 0,Y 474.614,Z 275.674,A -85,B 0,C 180,E1 -7152.934,E2 -7152.934} C_VEL
LIN {X 0,Y 474.608,Z 275.674,A -85,B 0,C 180,E1 -7155.895,E2 -7155.895} C_VEL
LIN {X 0,Y 474.626,Z 275.672,A -85,B 0,C 180,E1 -7159.04,E2 -7159.04} C_VEL
LIN {X 0,Y 474.608,Z 275.674,A -85,B 0,C 180,E1 -7161.704,E2 -7161.704} C_VEL
LIN {X 0,Y 474.627,Z 275.674,A -85,B 0,C 180,E1 -7164.726,E2 -7164.726} C_VEL
LIN {X 0,Y 474.633,Z 275.669,A -85,B 0,C 180,E1 -7167.787,E2 -7167.787} C_VEL
LIN {X 0,Y 474.622,Z 275.678,A -85,B 0,C 180,E1 -7170.884,E2 -7170.884} C_VEL
LIN {X 0,Y 474.659,Z 275.67,A -85,B 0,C 180,E1 -7173.628,E2 -7173.628} C_VEL
LIN {X 0,Y 474.633,Z 275.672,A -85,B 0,C 180,E1 -7176.641,E2 -7176.641} C_VEL
LIN {X 0,Y 474.652,Z 275.668,A -85,B 0,C 180,E1 -7180.089,E2 -7180.089} C_VEL
LIN {X 0,Y 474.645,Z 275.67,A -85,B 0,C 180,E1 -7182.774,E2 -7182.774} C_VEL
LIN {X 0,Y 474.646,Z 275.672,A -85,B 0,C 180,E1 -7185.421,E2 -7185.421} C_VEL
LIN {X 0,Y 474.701,Z 275.662,A -85,B 0,C 180,E1 -7188.037,E2 -7188.037} C_VEL
LIN {X 0,Y 474.724,Z 275.659,A -85,B 0,C 180,E1 -7191.486,E2 -7191.486} C_VEL
LIN {X 0,Y 474.779,Z 275.653,A -85,B 0,C 180,E1 -7194.052,E2 -7194.052} C_VEL
LIN {X 0,Y 474.892,Z 275.631,A -85,B 0,C 180,E1 -7197.455,E2 -7197.455} C_VEL
LIN {X 0,Y 474.909,Z 275.637,A -85,B 0,C 180,E1 -7200,E2 -7200} C_VEL
LIN {X 0,Y 474.891,Z 275.64,A -85,B 0,C 180,E1 -7202.544,E2 -7202.544} C_VEL
LIN {X 0,Y 474.778,Z 275.651,A -85,B 0,C 180,E1 -7205.947,E2 -7205.947} C_VEL
LIN {X 0,Y 474.725,Z 275.662,A -85,B 0,C 180,E1 -7208.513,E2 -7208.513} C_VEL
LIN {X 0,Y 474.701,Z 275.658,A -85,B 0,C 180,E1 -7211.962,E2 -7211.962} C_VEL
LIN {X 0,Y 474.697,Z 275.664,A -85,B 0,C 180,E1 -7215.456,E2 -7215.456} C_VEL
LIN {X 0,Y 474.662,Z 275.674,A -85,B 0,C 180,E1 -7219.01,E2 -7219.01} C_VEL
LIN {X 0,Y 474.585,Z 275.677,A -85,B 0,C 180,E1 -7221.729,E2 -7221.729} C_VEL
LIN {X 0,Y 474.656,Z 275.673,A -85,B 0,C 180,E1 -7224.493,E2 -7224.493} C_VEL
LIN {X 0,Y 474.678,Z 275.669,A -85,B 0,C 180,E1 -7227.334,E2 -7227.334} C_VEL
LIN {X 0,Y 474.602,Z 275.678,A -85,B 0,C 180,E1 -7230.23,E2 -7230.23} C_VEL
LIN {X 0,Y 474.64,Z 275.677,A -85,B 0,C 180,E1 -7233.22,E2 -7233.22} C_VEL
LIN {X 0,Y 474.59,Z 275.68,A -85,B 0,C 180,E1 -7236.323,E2 -7236.323} C_VEL
LIN {X 0,Y 474.624,Z 275.676,A -85,B 0,C 180,E1 -7239.648,E2 -7239.648} C_VEL
LIN {X 0,Y 474.612,Z 275.682,A -85,B 0,C 180,E1 -7242.934,E2 -7242.934} C_VEL
LIN {X 0,Y 474.612,Z 275.677,A -85,B 0,C 180,E1 -7245.896,E2 -7245.896} C_VEL
LIN {X 0,Y 474.63,Z 275.678,A -85,B 0,C 180,E1 -7249.04,E2 -7249.04} C_VEL
LIN {X 0,Y 474.607,Z 275.677,A -85,B 0,C 180,E1 -7251.704,E2 -7251.704} C_VEL
LIN {X 0,Y 474.622,Z 275.671,A -85,B 0,C 180,E1 -7254.726,E2 -7254.726} C_VEL
LIN {X 0,Y 474.657,Z 275.766,A -85,B 0,C 180,E1 -7257.173,E2 -7257.173} C_VEL
LIN {X 0,Y 480.117,Z 293.423,A -85,B 0,C 180,E1 -7259.524,E2 -7259.524} C_VEL
LIN {X 0,Y 482.355,Z 301.159,A -85,B 0,C 180,E1 -7260.512,E2 -7260.512} C_VEL
LIN {X 0,Y 482.419,Z 305.07,A -85,B 0,C 180,E1 -7260.937,E2 -7260.937} C_VEL
LIN {X 0,Y 482.104,Z 309.426,A -85,B 0,C 180,E1 -7261.387,E2 -7261.387} C_VEL
LIN {X 0,Y 486.302,Z 333.113,A -85,B 0,C 180,E1 -7262.051,E2 -7262.051} C_VEL
LIN {X 0,Y 484.681,Z 460.02,A -85,B 0,C 180,E1 -7264.015,E2 -7264.015} C_VEL
LIN {X 0,Y 483.885,Z 517.674,A -85,B 0,C 180,E1 -7264.926,E2 -7264.926} C_VEL
LIN {X 0,Y 483.339,Z 532.973,A -85,B 0,C 180,E1 -7265.318,E2 -7265.318} C_VEL
LIN {X 0,Y 482.613,Z 548.85,A -85,B 0,C 180,E1 -7265.88,E2 -7265.88} C_VEL
LIN {X 0,Y 481.738,Z 564.06,A -85,B 0,C 180,E1 -7266.575,E2 -7266.575} C_VEL
LIN {X 0,Y 480.786,Z 578.863,A -85,B 0,C 180,E1 -7267.424,E2 -7267.424} C_VEL
LIN {X 0,Y 479.73,Z 592.908,A -85,B 0,C 180,E1 -7268.403,E2 -7268.403} C_VEL
LIN {X 0,Y 478.643,Z 607.412,A -85,B 0,C 180,E1 -7269.613,E2 -7269.613} C_VEL
LIN {X 0,Y 477.601,Z 620.331,A -85,B 0,C 180,E1 -7270.888,E2 -7270.888} C_VEL
LIN {X 0,Y 476.744,Z 631.577,A -85,B 0,C 180,E1 -7272.189,E2 -7272.189} C_VEL
LIN {X 0,Y 475.91,Z 642.87,A -85,B 0,C 180,E1 -7273.716,E2 -7273.716} C_VEL
LIN {X 0,Y 475.271,Z 652.433,A -85,B 0,C 180,E1 -7275.222,E2 -7275.222} C_VEL
LIN {X 0,Y 474.718,Z 661.803,A -85,B 0,C 180,E1 -7276.952,E2 -7276.952} C_VEL
LIN {X 0,Y 474.269,Z 670.485,A -85,B 0,C 180,E1 -7278.893,E2 -7278.893} C_VEL
LIN {X 0,Y 473.953,Z 678.176,A -85,B 0,C 180,E1 -7281.043,E2 -7281.043} C_VEL
LIN {X 0,Y 473.823,Z 684.03,A -85,B 0,C 180,E1 -7283.185,E2 -7283.185} C_VEL
LIN {X 0,Y 473.759,Z 687.453,A -85,B 0,C 180,E1 -7284.894,E2 -7284.894} C_VEL
LIN {X 0,Y 473.773,Z 689.943,A -85,B 0,C 180,E1 -7286.598,E2 -7286.598} C_VEL
LIN {X 0,Y 473.689,Z 691.345,A -85,B 0,C 180,E1 -7288.3,E2 -7288.3} C_VEL
LIN {X 0,Y 473.665,Z 691.873,A -85,B 0,C 180,E1 -7290,E2 -7290} C_VEL
LIN {X 0,Y 473.689,Z 691.344,A -85,B 0,C 180,E1 -7291.7,E2 -7291.7} C_VEL
LIN {X 0,Y 473.773,Z 689.941,A -85,B 0,C 180,E1 -7293.402,E2 -7293.402} C_VEL
LIN {X 0,Y 473.759,Z 687.453,A -85,B 0,C 180,E1 -7295.106,E2 -7295.106} C_VEL
LIN {X 0,Y 473.823,Z 684.033,A -85,B 0,C 180,E1 -7296.815,E2 -7296.815} C_VEL
LIN {X 0,Y 473.953,Z 678.179,A -85,B 0,C 180,E1 -7298.957,E2 -7298.957} C_VEL
LIN {X 0,Y 474.269,Z 670.485,A -85,B 0,C 180,E1 -7301.107,E2 -7301.107} C_VEL
LIN {X 0,Y 474.718,Z 661.803,A -85,B 0,C 180,E1 -7303.048,E2 -7303.048} C_VEL
LIN {X 0,Y 475.27,Z 652.434,A -85,B 0,C 180,E1 -7304.778,E2 -7304.778} C_VEL
LIN {X 0,Y 475.934,Z 642.799,A -85,B 0,C 180,E1 -7306.294,E2 -7306.294} C_VEL
LIN {X 0,Y 476.762,Z 631.574,A -85,B 0,C 180,E1 -7307.811,E2 -7307.811} C_VEL
LIN {X 0,Y 477.712,Z 619.346,A -85,B 0,C 180,E1 -7309.219,E2 -7309.219} C_VEL
LIN {X 0,Y 478.74,Z 606.109,A -85,B 0,C 180,E1 -7310.506,E2 -7310.506} C_VEL
LIN {X 0,Y 479.757,Z 592.898,A -85,B 0,C 180,E1 -7311.596,E2 -7311.596} C_VEL
LIN {X 0,Y 480.772,Z 578.885,A -85,B 0,C 180,E1 -7312.574,E2 -7312.574} C_VEL
LIN {X 0,Y 481.763,Z 563.035,A -85,B 0,C 180,E1 -7313.48,E2 -7313.48} C_VEL
LIN {X 0,Y 482.664,Z 547.524,A -85,B 0,C 180,E1 -7314.175,E2 -7314.175} C_VEL
LIN {X 0,Y 483.377,Z 531.104,A -85,B 0,C 180,E1 -7314.737,E2 -7314.737} C_VEL
LIN {X 0,Y 483.973,Z 513.446,A -85,B 0,C 180,E1 -7315.15,E2 -7315.15} C_VEL
LIN {X 0,Y 486.405,Z 333.938,A -85,B 0,C 180,E1 -7317.927,E2 -7317.927} C_VEL
LIN {X 0,Y 482.07,Z 309.451,A -85,B 0,C 180,E1 -7318.609,E2 -7318.609} C_VEL
LIN {X 0,Y 482.505,Z 303.058,A -85,B 0,C 180,E1 -7319.272,E2 -7319.272} C_VEL
LIN {X 0,Y 482.379,Z 301.142,A -85,B 0,C 180,E1 -7319.486,E2 -7319.486} C_VEL
LIN {X 0,Y 476.682,Z 282.324,A -85,B 0,C 180,E1 -7321.937,E2 -7321.937} C_VEL
LIN {X 0,Y 474.621,Z 275.673,A -85,B 0,C 180,E1 -7322.844,E2 -7322.844} C_VEL
LIN {X 0,Y 474.612,Z 275.68,A -85,B 0,C 180,E1 -7325.469,E2 -7325.469} C_VEL
LIN {X 0,Y 474.609,Z 275.677,A -85,B 0,C 180,E1 -7328.457,E2 -7328.457} C_VEL
LIN {X 0,Y 474.63,Z 275.676,A -85,B 0,C 180,E1 -7330.96,E2 -7330.96} C_VEL
LIN {X 0,Y 474.613,Z 275.673,A -85,B 0,C 180,E1 -7334.104,E2 -7334.104} C_VEL
LIN {X 0,Y 474.612,Z 275.677,A -85,B 0,C 180,E1 -7337.066,E2 -7337.066} C_VEL
LIN {X 0,Y 474.615,Z 275.67,A -85,B 0,C 180,E1 -7340.354,E2 -7340.354} C_VEL
LIN {X 0,Y 474.589,Z 275.677,A -85,B 0,C 180,E1 -7343.677,E2 -7343.677} C_VEL
LIN {X 0,Y 474.64,Z 275.672,A -85,B 0,C 180,E1 -7346.78,E2 -7346.78} C_VEL
LIN {X 0,Y 474.602,Z 275.674,A -85,B 0,C 180,E1 -7349.77,E2 -7349.77} C_VEL
LIN {X 0,Y 474.694,Z 275.665,A -85,B 0,C 180,E1 -7352.68,E2 -7352.68} C_VEL
LIN {X 0,Y 474.656,Z 275.672,A -85,B 0,C 180,E1 -7355.507,E2 -7355.507} C_VEL
LIN {X 0,Y 474.667,Z 275.66,A -85,B 0,C 180,E1 -7359.185,E2 -7359.185} C_VEL
LIN {X 0,Y 474.653,Z 275.668,A -85,B 0,C 180,E1 -7361.884,E2 -7361.884} C_VEL
LIN {X 0,Y 474.697,Z 275.664,A -85,B 0,C 180,E1 -7364.544,E2 -7364.544} C_VEL
LIN {X 0,Y 474.702,Z 275.658,A -85,B 0,C 180,E1 -7368.038,E2 -7368.038} C_VEL
LIN {X 0,Y 474.725,Z 275.657,A -85,B 0,C 180,E1 -7371.487,E2 -7371.487} C_VEL
LIN {X 0,Y 474.778,Z 275.64,A -85,B 0,C 180,E1 -7374.053,E2 -7374.053} C_VEL
LIN {X 0,Y 474.892,Z 275.641,A -85,B 0,C 180,E1 -7377.456,E2 -7377.456} C_VEL
LIN {X 0,Y 474.909,Z 275.626,A -85,B 0,C 180,E1 -7380,E2 -7380} C_VEL
LIN {X 0,Y 474.892,Z 275.633,A -85,B 0,C 180,E1 -7382.545,E2 -7382.545} C_VEL
LIN {X 0,Y 474.768,Z 275.652,A -85,B 0,C 180,E1 -7385.948,E2 -7385.948} C_VEL
LIN {X 0,Y 474.725,Z 275.645,A -85,B 0,C 180,E1 -7388.514,E2 -7388.514} C_VEL
LIN {X 0,Y 474.702,Z 275.663,A -85,B 0,C 180,E1 -7391.963,E2 -7391.963} C_VEL
